// ── Aggregate readiness / faults ──────────────────────────────────────────────
allReady :=
    upperMasterReady AND upperSlave1VfdReady AND upperSlave2VfdReady AND
    lowerMasterReady AND lowerSlave1VfdReady AND lowerSlave2VfdReady;

anyFault :=
    groupFault OR
    upperMasterVfdFaultFeedback OR upperSlave1VfdFaultFeedback OR upperSlave2VfdFaultFeedback OR
    lowerMasterVfdFaultFeedback OR lowerSlave1VfdFaultFeedback OR lowerSlave2VfdFaultFeedback;

// ── Near-zero checks (unit must match your speed signals) ─────────────────────
speedsNearZero :=
    (ABS(upperMasterSpeedFeedback) <= speedZeroThresholdPct) AND
    (ABS(upperSlave1SpeedFeedback) <= speedZeroThresholdPct) AND
    (ABS(upperSlave2SpeedFeedback) <= speedZeroThresholdPct) AND
    (ABS(lowerMasterSpeedFeedback) <= speedZeroThresholdPct) AND
    (ABS(lowerSlave1SpeedFeedback) <= speedZeroThresholdPct) AND
    (ABS(lowerSlave2SpeedFeedback) <= speedZeroThresholdPct);

// Masters’ references near zero (backup condition)
refsNearZero :=
    (ABS(upperMasterDriveSpeedRefRPM) <= epsRefPct) AND
    (ABS(lowerMasterDriveSpeedRefRPM) <= epsRefPct);

// ── State machine ─────────────────────────────────────────────────────────────
CASE state OF
    0: // IDLE
        deviceState := 'IDLE';
        rampReset   := TRUE;

        // Ensure outputs are safe
        upperMasterDriveEnable := FALSE;
        upperSlave1DriveEnable := FALSE;
        upperSlave2DriveEnable := FALSE;
        lowerMasterDriveEnable := FALSE;
        lowerSlave1DriveEnable := FALSE;
        lowerSlave2DriveEnable := FALSE;

        IF rStart AND NOT anyFault THEN
            state := 1;
        END_IF

    1: // ENABLE_DRIVES
        deviceState := 'ENABLE_DRIVES';
        rampReset   := TRUE;

        // Enable all six drives
        upperMasterDriveEnable := TRUE;
        upperSlave1DriveEnable := TRUE;
        upperSlave2DriveEnable := TRUE;
        lowerMasterDriveEnable := TRUE;
        lowerSlave1DriveEnable := TRUE;
        lowerSlave2DriveEnable := TRUE;

        // Start enable wait timer
        instTONEnableWait(IN := TRUE, PT := enableTimeout);

        IF rStop OR stopGroup THEN
            instTONEnableWait(IN := FALSE);
            state := 5; // go to stopping
        ELSE
            state := 2; // proceed to wait feedback
        END_IF

    2: // WAIT_ENABLE_FEEDBACK
        deviceState := 'WAIT_ENABLE_FEEDBACK';
        rampReset   := TRUE;

        // Keep enables on while waiting
        upperMasterDriveEnable := TRUE;
        upperSlave1DriveEnable := TRUE;
        upperSlave2DriveEnable := TRUE;
        lowerMasterDriveEnable := TRUE;
        lowerSlave1DriveEnable := TRUE;
        lowerSlave2DriveEnable := TRUE;

        instTONEnableWait(IN := TRUE, PT := enableTimeout);

        IF anyFault THEN
            instTONEnableWait(IN := FALSE);
            state := 10; // FAULT
        ELSIF rStop OR stopGroup THEN
            instTONEnableWait(IN := FALSE);
            state := 5; // STOPPING
        ELSIF allReady THEN
            instTONEnableWait(IN := FALSE);
            state := 3; // RAMP_ENABLE
        ELSIF instTONEnableWait.Q THEN
            instTONEnableWait(IN := FALSE);
            state := 10; // fault: no enable feedback in time
        END_IF

    3: // RAMP_ENABLE (single-cycle gate to release ramp)
        deviceState := 'RAMP_ENABLE';
        rampReset   := FALSE; // release ramp now

        // Keep enables on
        upperMasterDriveEnable := TRUE;
        upperSlave1DriveEnable := TRUE;
        upperSlave2DriveEnable := TRUE;
        lowerMasterDriveEnable := TRUE;
        lowerSlave1DriveEnable := TRUE;
        lowerSlave2DriveEnable := TRUE;

        IF rStop OR stopGroup THEN
            state := 5;
        ELSE	
		
            state := 4; // RUN
					
        END_IF

    4: // RUN
        deviceState := SEL(groupSpeedAutoMan, 'RUN (Manual)', 'RUN (Auto)');
        rampReset   := FALSE;

        // Keep enables on during run
        upperMasterDriveEnable := TRUE;
        upperSlave1DriveEnable := TRUE;
        upperSlave2DriveEnable := TRUE;
        lowerMasterDriveEnable := TRUE;
        lowerSlave1DriveEnable := TRUE;
        lowerSlave2DriveEnable := TRUE;

        IF anyFault THEN
            state := 10; // FAULT
        ELSIF rStop OR stopGroup THEN
            state := 5;  // STOPPING
        END_IF

    5: // STOPPING (controlled decel)
        deviceState := 'STOPPING';
        rampReset   := FALSE; // allow ramp to drive refs down

        // Keep enables TRUE for controlled decel
        upperMasterDriveEnable := TRUE;
        upperSlave1DriveEnable := TRUE;
        upperSlave2DriveEnable := TRUE;
        lowerMasterDriveEnable := TRUE;
        lowerSlave1DriveEnable := TRUE;
        lowerSlave2DriveEnable := TRUE;

        // Optional: stop timeout (enable if you want a hard cutoff)
        // instTONStopWait(IN := TRUE, PT := stopTimeout);

        // Exit when speeds≈0 and refs≈0
        IF anyFault THEN
            // instTONStopWait(IN := FALSE);
            state := 10;

        ELSIF speedsNearZero AND refsNearZero THEN
            // Disable all drives
            upperMasterDriveEnable := FALSE;
            upperSlave1DriveEnable := FALSE;
            upperSlave2DriveEnable := FALSE;
            lowerMasterDriveEnable := FALSE;
            lowerSlave1DriveEnable := FALSE;
            lowerSlave2DriveEnable := FALSE;

            // instTONStopWait(IN := FALSE);
            state := 0; // IDLE

        ELSIF instTONStopWait.Q THEN
            // Timeout path → force disable then fault
            upperMasterDriveEnable := FALSE;
            upperSlave1DriveEnable := FALSE;
            upperSlave2DriveEnable := FALSE;
            lowerMasterDriveEnable := FALSE;
            lowerSlave1DriveEnable := FALSE;
            lowerSlave2DriveEnable := FALSE;

            instTONStopWait(IN := FALSE);
            state := 10;
        END_IF

    10: // FAULT
        deviceState := 'FAULT';
        rampReset   := TRUE; // force ramp outputs to zero

        // Disable all drives
        upperMasterDriveEnable := FALSE;
        upperSlave1DriveEnable := FALSE;
        upperSlave2DriveEnable := FALSE;
        lowerMasterDriveEnable := FALSE;
        lowerSlave1DriveEnable := FALSE;
        lowerSlave2DriveEnable := FALSE;

        // Return to IDLE when faults clear and start released
        IF (NOT anyFault) AND (NOT startGroup) THEN
            state := 0;
        END_IF
END_CASE
END_METHOD

// 2) REFERENCE GENERATOR
// Applies:
//   - groupSpeedOffset: added to ALL motors in this drying section (via ratio)
//   - uperAndLowerSpeedOffset: additional bias between UPPER and LOWER groups only
METHOD _ReferenceGenerator
VAR
    // ---------- Limits & helpers ----------
    headroomEpsPct      : REAL := 0.20;     // anti-chatter near saturation (100%)
    offsetPct           : REAL;             // slave speed offset as ratio (e.g., 10% -> 0.10)
    denom               : REAL;             // gear + offset denominator guard
    maxMasterBySlave    : REAL;             // master % at which a slave would hit 100%
    allowedCapPct       : REAL;             // master upward cap (prevents slave > 100%)
    cmdSpeedMPM         : REAL;             // selected command speed (m/min)
    targetRPM           : REAL;             // 0..100 scaled line reference before ramp

    // ---------- Freeze upward overrun ----------
    currMasterPct       : REAL;             // current ramp output for master (%)
    currSlavePct        : REAL;             // current synthetic slave (%), for freeze check

    // ---------- Group offsets ----------
    groupDeltaRatioAll  : REAL;             // = 1 + (groupSpeedOffset / 100) → applies to ALL motors
    upperLowerBiasRatio : REAL;             // = 1 + (uperAndLowerSpeedOffset / 100) → LOWER only

    // ---------- Convenience ----------
    baseMasterRefRPM    : REAL;             // common master reference after ramp/cap (pre-offsets)
    baseCmdSpeedMPM     : REAL;             // base command (auto/manual, pre-recover)

//	masterMaxSpeedMPM : REAL;

	PI : REAL := 3.14159265359;
	
	k_pi_per_1000 : REAL := 0.00314159265358979323846264338328;
	
END_VAR
//==============================================================
// Calculate max output speed in MPM
//==============================================================
masterMaxSpeedMPM := groupMasterMaxSpeedRPM * (PI * upperMasterDiameter) / 1000.0;


//==============================================================
// 1) Determine base speed source (auto or manual)
//==============================================================
IF groupSpeedAutoMan THEN
    baseCmdSpeedMPM := groupAutoSpeedMPM * interGroupGearRatio; // Auto reference (calibrated)
ELSE
    baseCmdSpeedMPM := groupManualSpeedMPM;                      // Manual reference (raw)
END_IF;


//==============================================================
// 2) Apply "Recover" temporary speed bump
//==============================================================
IF groupRecoverSpeedCmd THEN
    cmdSpeedMPM := baseCmdSpeedMPM + groupRecoverIncrement;     // Apply recover bump
ELSE
    cmdSpeedMPM := baseCmdSpeedMPM;                             // Normal operation
END_IF;


//==============================================================
// 3) Scale to target RPM for the drives 
//==============================================================
targetRPM := _Scale(
    X    := cmdSpeedMPM,
    I_LO := 0.0,          I_HI := masterMaxSpeedMPM,
    O_LO := 0.0,          O_HI := groupMasterMaxSpeedRPM);
	

//==============================================================
// 4) During STOPPING set target to 0 (still ramp down); otherwise track target
//==============================================================
IF state = 5 THEN
    rampTargetRPM := 0.0;
ELSE
    rampTargetRPM := targetRPM;
END_IF;


//==============================================================
// 5) Ramp (common line reference for this drying section)
//==============================================================
useRamp := (ABS(rampTargetRPM - instFB_Gen_SRamp.Y) >= 2.0);

instFB_Gen_SRamp(
    X          := rampTargetRPM,
    A_UP       := MAX(0.0, rampRate),
    A_DN       := -MAX(0.0, rampRate),
    VU_MAX     := 1000.0,
    VD_MAX     := -1000.0,
    LIMIT_HIGH := groupMasterMaxSpeedRPM,
    RST        := rampReset);

IF useRamp THEN
    baseMasterRefRPM := instFB_Gen_SRamp.Y;
ELSE
    baseMasterRefRPM := rampTargetRPM;
END_IF;


//==============================================================
// 6) Operator-adjustable groupSpeedOffset using TUNE2
//==============================================================
instTUNE2_GroupSpeedDiference(
    SET     := FALSE,
    SU      := groupSpeedDifInc,
    SD      := groupSpeedDifDec,
    RST     := FALSE,
    SS      := 0.1,
    FS      := 0.0,
    LIMIT_L := groupSpeedDifLimLow,
    LIMIT_H := groupSpeedDifLimHigh,
    Y       => groupSpeedOffset);

groupDeltaRatioAll  := 1.0 + (groupSpeedOffset * 0.01);
upperLowerBiasRatio := 1.0 + (upperAndLowerSpeedOffset * 0.01);


//==============================================================
// 7) MASTER references and slave ratios
//==============================================================
upperMasterDriveSpeedRefRPM := baseMasterRefRPM * groupDeltaRatioAll;

upperSlave1DriveSpeedRefRPM := upperMasterDriveSpeedRefRPM * upperToUpperSlave1Ratio;
upperSlave2DriveSpeedRefRPM := upperMasterDriveSpeedRefRPM * upperToUpperSlave2Ratio;

lowerMasterDriveSpeedRefRPM := upperMasterDriveSpeedRefRPM * upperToLowerMasterRatio;
lowerSlave1DriveSpeedRefRPM := lowerMasterDriveSpeedRefRPM * lowerToLowerSlave1Ratio;
lowerSlave2DriveSpeedRefRPM := lowerMasterDriveSpeedRefRPM * lowerToLowerSlave2Ratio;


//==============================================================
// 8) Convert drive RPM references to surface speeds in MPM
//==============================================================
upperMasterSpeedSetpointMPM := upperMasterDriveSpeedRefRPM * upperMasterDiameter * PI / 1000.0;
upperSlave1SpeedSetpointMPM := upperSlave1DriveSpeedRefRPM * upperSlave1Diameter * PI / 1000.0;
upperSlave2SpeedSetpointMPM := upperSlave2DriveSpeedRefRPM * upperSlave2Diameter * PI / 1000.0;

lowerMasterSpeedSetpointMPM := lowerMasterDriveSpeedRefRPM * lowerMasterDiameter * PI / 1000.0;
lowerSlave1SpeedSetpointMPM := lowerSlave1DriveSpeedRefRPM * lowerSlave1Diameter * PI / 1000.0;
lowerSlave2SpeedSetpointMPM := lowerSlave2DriveSpeedRefRPM * lowerSlave2Diameter * PI / 1000.0;
END_METHOD

METHOD PRIVATE _Scale : REAL
VAR_INPUT
    X    : REAL;
    I_LO : REAL;
    I_HI : REAL;
    O_LO : REAL;
    O_HI : REAL;
END_VAR
IF I_LO = I_HI THEN
	_Scale := O_LO;
ELSE
	_Scale := (O_HI - O_LO) / (I_HI - I_LO) * (LIMIT(I_LO, X, I_HI) - I_LO) + O_LO;
END_IF;
END_METHOD

METHOD PRIVATE _SpeedDifferenceCheck
VAR
    diffUpper : REAL; // max |Master - Slave| in UPPER group
    diffLower : REAL; // max |Master - Slave| in LOWER group
    diffMax   : REAL; // worst-case across both groups
END_VAR

(*
// ── Compare only within each group: Master ↔ Slaves (ignore cross-group) ──────
// UPPER group (Master vs Slave1, Master vs Slave2)
diffUpper :=
    MAX(
        ABS(upperMasterSpeedMPMFilteredDisplay - upperSlave1SpeedMPMFilteredDisplay),
        ABS(upperMasterSpeedMPMFilteredDisplay - upperSlave2SpeedMPMFilteredDisplay)
    );

// LOWER group (Master vs Slave1, Master vs Slave2)
diffLower :=
    MAX(
        ABS(lowerMasterSpeedMPMFilteredDisplay - lowerSlave1SpeedMPMFilteredDisplay),
        ABS(lowerMasterSpeedMPMFilteredDisplay - lowerSlave2SpeedMPMFilteredDisplay)
    );

// Pick worst intra-group deviation and expose for diagnostics/HMI
diffMax := MAX(diffUpper, diffLower);
currentSpeedDifence := diffMax;

// ── Trip logic with delay (debounce) ───────────────────────────────────────────
instTONSpeedDifDelay(
    IN := (diffMax > speedDiferenceLimit),
    PT := T#2s
);

IF instTONSpeedDifDelay.Q THEN
    state := 10; // FAULT
    deviceState := 'FAULT: Intra-group speed difference exceeded';
END_IF
*)
END_METHOD

METHOD _StateDisplay
VAR_INPUT
END_VAR

// ──────────────────────────────────────────────────────────────────────────────
// _StateDisplay
// Maps the internal machine "state" to a compact HMI status code and derives
// per-drive motor status codes from VFD signals.
//
// statusCode / masterStatusCode / slaveStatusCode legend:
//   0 = Idle, 1 = Starting, 2 = Running, 3 = Fault
//
// Machine "state" groups:
//   0 = IDLE, 1 = ENABLE, 2 = WAIT_EN, 3 = RAMP_EN, 4 = RUN, 5 = STOPPING, 10 = FAULT
// Priority rule (for motors): Fault > Running > Starting > Idle
// ──────────────────────────────────────────────────────────────────────────────
VAR CONSTANT
    STATUS_IDLE     : INT := 0;
    STATUS_STARTING : INT := 1;
    STATUS_RUNNING  : INT := 1;
    STATUS_FAULT    : INT := 2;
END_VAR
// ─────────────── Group machine states into a single HMI statusCode ───────────
CASE state OF
    10: // FAULT
        statusCode := STATUS_FAULT;
    4:  // RUN
        statusCode := STATUS_RUNNING;
    1, 2, 3: // ENABLE / WAIT_EN / RAMP_EN
        statusCode := STATUS_STARTING;
ELSE // IDLE, STOPPING, or any other
        statusCode := STATUS_IDLE;
END_CASE;


// ─────────────── Per-drive status (priority: Fault > Running > Starting > Idle) ───────────────
// UPPER — MASTER
IF upperMasterVfdFaultFeedback THEN
    upperMasterStatusCode := STATUS_FAULT;
ELSIF upperMasterVfdRunFeedback THEN
    upperMasterStatusCode := STATUS_RUNNING;
ELSIF upperMasterDriveEnable THEN
    upperMasterStatusCode := STATUS_STARTING;
ELSE
    upperMasterStatusCode := STATUS_IDLE;
END_IF;

// UPPER — SLAVE 1
IF upperSlave1VfdFaultFeedback THEN
    upperSlave1StatusCode := STATUS_FAULT;
ELSIF upperSlave1VfdRunFeedback THEN
    upperSlave1StatusCode := STATUS_RUNNING;
ELSIF upperSlave1DriveEnable THEN
    upperSlave1StatusCode := STATUS_STARTING;
ELSE
    upperSlave1StatusCode := STATUS_IDLE;
END_IF;

// UPPER — SLAVE 2
IF upperSlave2VfdFaultFeedback THEN
    upperSlave2StatusCode := STATUS_FAULT;
ELSIF upperSlave2VfdRunFeedback THEN
    upperSlave2StatusCode := STATUS_RUNNING;
ELSIF upperSlave2DriveEnable THEN
    upperSlave2StatusCode := STATUS_STARTING;
ELSE
    upperSlave2StatusCode := STATUS_IDLE;
END_IF;

// LOWER — MASTER
IF lowerMasterVfdFaultFeedback THEN
    lowerMasterStatusCode := STATUS_FAULT;
ELSIF lowerMasterVfdRunFeedback THEN
    lowerMasterStatusCode := STATUS_RUNNING;
ELSIF lowerMasterDriveEnable THEN
    lowerMasterStatusCode := STATUS_STARTING;
ELSE
    lowerMasterStatusCode := STATUS_IDLE;
END_IF;

// LOWER — SLAVE 1
IF lowerSlave1VfdFaultFeedback THEN
    lowerSlave1StatusCode := STATUS_FAULT;
ELSIF lowerSlave1VfdRunFeedback THEN
    lowerSlave1StatusCode := STATUS_RUNNING;
ELSIF lowerSlave1DriveEnable THEN
    lowerSlave1StatusCode := STATUS_STARTING;
ELSE
    lowerSlave1StatusCode := STATUS_IDLE;
END_IF;

// LOWER — SLAVE 2
IF lowerSlave2VfdFaultFeedback THEN
    lowerSlave2StatusCode := STATUS_FAULT;
ELSIF lowerSlave2VfdRunFeedback THEN
    lowerSlave2StatusCode := STATUS_RUNNING;
ELSIF lowerSlave2DriveEnable THEN
    lowerSlave2StatusCode := STATUS_STARTING;
ELSE
    lowerSlave2StatusCode := STATUS_IDLE;
END_IF;
END_METHOD

METHOD _SteamPressureControl
VAR_INPUT
END_VAR

//────────────────────────────────────────────────────────────
// PID — Steam Pressure Control
//────────────────────────────────────────────────────────────
instCTRL_PID_TemperatureController(
    ACT := steamPressureFeedback,                          // Real-time feedback (PV)
    SET := SEL(steamPressureAutoMan,                       // Setpoint selection
               steamPressureManualSetpoint,                // Manual setpoint
               steamPressureAutoSetpoint),                 // Auto setpoint
    MAN := steamPressureAutoMan = FALSE,                   // Manual mode when AutoMan is FALSE
    M_I := steamPressureManualSetpoint,                    // Tracks manual setpoint
    RST := FALSE,                                          // No reset
    KP  := steamPressureKp,                               
    TN  := steamPressureTn,                               
    TV  := steamPressureTv,                               
    LL  := 0.0,                                            // Output lower limit
    LH  := 100.0,                                          // Output upper limit [%]
    Y   => steamPressureControllerOutput                   // PID output
);
END_METHOD

METHOD PRIVATE _TorqueReference
VAR
    // UPPER
    rawTorqueUpper      : REAL;
    filteredTorqueUpper : REAL;
    capMasterUpper      : REAL; // ≤ master, ≤ global max
    baseLimitUpper      : REAL; // (master + offset) capped by master
    directTorqueUpper   : REAL; // direct write portion
    avgTorqueUpper      : REAL;
    trimUp              : REAL; // PID top-up (≥0)

    // LOWER
    rawTorqueLower      : REAL;
    filteredTorqueLower : REAL;
    capMasterLower      : REAL;
    baseLimitLower      : REAL;
    directTorqueLower   : REAL;
    avgTorqueLower      : REAL;
    trimLo              : REAL;
END_VAR


// ── UPPER ─────────────────────────────────────────────────────────────────────
rawTorqueUpper := upperMasterTorqueFeedback;
instsFT_PT1UpperTorqueFilter( in := rawTorqueUpper, 
							   T := torqueFilterTime, 
							   K := 1.0, 
							   out => filteredTorqueUpper );
							   

// Master cap and base limit (never exceed master)
capMasterUpper := LIMIT(torqueLimitMinPct, filteredTorqueUpper, torqueLimitMaxPct);
baseLimitUpper := MIN(
    capMasterUpper,
    LIMIT(torqueLimitMinPct, filteredTorqueUpper + slaveTorqueOfsset, torqueLimitMaxPct)
);

IF NOT enableTorquePid THEN
    upperSlave1DriveTorqueRefPct := capMasterUpper;
    upperSlave2DriveTorqueRefPct := capMasterUpper;
ELSE
    directTorqueUpper := LIMIT(torqueLimitMinPct, baseLimitUpper - torqueTrimLimit, capMasterUpper);
    avgTorqueUpper    := 0.5 * (upperSlave1TorqueFeedback + upperSlave2TorqueFeedback);

    instCTRL_PID_UpperTorqueTrim(
        ACT := avgTorqueUpper,
        SET := baseLimitUpper,
        MAN := NOT enableTorquePid,   // manual when disabled (tracks 0)
        M_I := 0.0,
        RST := FALSE,
        KP  := torqueCtrlKp,
        TN  := torqueCtrlTn,
        TV  := torqueCtrlTv,
        LL  := 0.0,                   // unipolar: only add
        LH  := torqueTrimLimit,
        Y   => trimUp
    );

    upperSlave1DriveTorqueRefPct := LIMIT(torqueLimitMinPct, directTorqueUpper + trimUp, capMasterUpper);
    upperSlave2DriveTorqueRefPct := LIMIT(torqueLimitMinPct, directTorqueUpper + trimUp, capMasterUpper);
END_IF;


// ── LOWER ─────────────────────────────────────────────────────────────────────
rawTorqueLower := lowerMasterTorqueFeedback;
instsFT_PT1LowerTorqueFilter( in := rawTorqueLower, T := torqueFilterTime, K := 1.0, out => filteredTorqueLower );

capMasterLower := LIMIT(torqueLimitMinPct, filteredTorqueLower, torqueLimitMaxPct);
baseLimitLower := MIN(
    capMasterLower,
    LIMIT(torqueLimitMinPct, filteredTorqueLower + slaveTorqueOfsset, torqueLimitMaxPct)
);

IF NOT enableTorquePid THEN
    lowerSlave1DriveTorqueRefPct := capMasterLower;
    lowerSlave2DriveTorqueRefPct := capMasterLower;
ELSE
    directTorqueLower := LIMIT(torqueLimitMinPct, baseLimitLower - torqueTrimLimit, capMasterLower);
    avgTorqueLower    := 0.5 * (lowerSlave1TorqueFeedback + lowerSlave2TorqueFeedback);

    instCTRL_PID_LowerTorqueTrim(
        ACT := avgTorqueLower,
        SET := baseLimitLower,
        MAN := NOT enableTorquePid,
        M_I := 0.0,
        RST := FALSE,
        KP  := torqueCtrlKp,
        TN  := torqueCtrlTn,
        TV  := torqueCtrlTv,
        LL  := 0.0,
        LH  := torqueTrimLimit,
        Y   => trimLo
    );

    lowerSlave1DriveTorqueRefPct := LIMIT(torqueLimitMinPct, directTorqueLower + trimLo, capMasterLower);
    lowerSlave2DriveTorqueRefPct := LIMIT(torqueLimitMinPct, directTorqueLower + trimLo, capMasterLower);
END_IF;


// ── Safety (optional) ─────────────────────────────────────────────────────────
IF (state < 3) OR (state = 5) OR (state = 10) THEN
    upperSlave1DriveTorqueRefPct := 0.0;
    upperSlave2DriveTorqueRefPct := 0.0;
    lowerSlave1DriveTorqueRefPct := 0.0;
    lowerSlave2DriveTorqueRefPct := 0.0;
END_IF
END_METHOD

END_FUNCTION_BLOCK

// ---- Function Blocks/Rewinder/FB_RewinderControl_V1.TcPOU
FUNCTION_BLOCK FB_RewinderControl_V1
VAR_INPUT

    //==============================================================
    // ─────────────── BASIC COMMANDS / MACHINE INTERFACE ───────────────
    //==============================================================
    startCmd                    : BOOL;  // EN: Start rewinder command / PT: Comando de partida do rebobinador
    stopCmd                     : BOOL;  // EN: Stop rewinder command / PT: Comando de parada do rebobinador
	
	jogCmd						: BOOL;
  
	rewinderAutoMan            : BOOL;  // EN: Auto/Manual selector (FALSE = Manual) / PT: Seletor Auto/Manual (FALSE = Manual)

	
	rollEjectorFwCmd			: BOOL;
	rollEjectorRevCmd			: BOOL;
	
	
	
    //==============================================================
    // ─────────────── SPEED MONITORING / LIMITS ───────────────
    //==============================================================
    speedFeedBackMPM           : REAL;  // EN: Actual machine speed [m/min] / PT: Velocidade atual da máquina [m/min]
    groupMaxSpeed              : REAL;  // EN: Max allowed speed [m/min] / PT: Velocidade máxima permitida [m/min]

    //==============================================================
    // ─────────────── PRESS ROLL / NIP CONTROL ───────────────
    //==============================================================
    pressRollAutoMan           : BOOL;  // EN: Press roll Auto/Manual selector (FALSE = Manual) / PT: Seletor Auto/Manual do rolo de pressão (FALSE = Manual)
  
    pressRollManualSetpoint    : REAL;  // EN: Manual press roll setpoint / PT: Setpoint manual de posição/pressão do rolo de pressão
    //==============================================================
    // ─────────────── PRESS ROLL / NIP OUTPUTS ───────────────
    //==============================================================

    pressRollCmdUp             : BOOL;  // EN: Output command to open press roll / PT: Comando de abertura do rolo de pressão
    pressRollCmdDown           : BOOL;  // EN: Output command to close press roll / PT: Comando de fechamento do rolo de pressão

    //==============================================================
    // ─────────────── DIAMETER INPUTS ───────────────
    //==============================================================
    rewinderRollDiameter       : REAL;  // EN: Rewinder roll (winding) diameter [mm] / PT: Diâmetro do rolo rebobinado [mm]
    unwinderRollDiameter       : REAL;  // EN: Unwinder roll (payoff) diameter [mm] / PT: Diâmetro do rolo desbobinado [mm]

    //==============================================================
    // ─────────────── TENSION CONTROL ───────────────
    //==============================================================
    tensionSetpointN           : REAL;  // EN: Web tension setpoint [N] / PT: Setpoint de tensão da folha [N]
    tensionFeedbackN           : REAL;  // EN: Web tension feedback from load cell [N] / PT: Leitura de tensão da célula de carga [N]
    tensionControlEnable       : BOOL;  // EN: Enable tension control / PT: Habilita controle de tensão

    //==============================================================
    // ─────────────── ROLL LIMITS ───────────────
    //==============================================================
    maxRewinderDiameter        : REAL;  // EN: Max rewinder roll diameter [mm] / PT: Diâmetro máximo do rebobinador [mm]

    //==============================================================
    // ─────────────── SAFETY / INTERLOCKS ───────────────
    //==============================================================
    safetyCircuitOK            : BOOL;  // EN: Safety circuit healthy / PT: Circuito de segurança OK
    webBreakSensor             : BOOL;  // EN: Web break sensor triggered / PT: Sensor de ruptura de folha

    //==============================================================
    // ─────────────── SPEED REFERENCE INPUTS ───────────────
    //==============================================================
    rewinderAutoSpeedRefMPM    : REAL;  // EN: Auto speed reference (external) [m/min] / PT: Referência automática de velocidade [m/min]
    rewinderManualSpeedRefMPM  : REAL;  // EN: Manual speed reference [m/min] / PT: Referência manual de velocidade [m/min]
    rampRate                   : REAL := 0.01;  // EN: Ramp acceleration rate [%/s] / PT: Taxa de aceleração da rampa [%/s]
	
	
    //==============================================================
    // ─────────────── WEB GUIDING / EDGE CONTROL ───────────────
    //==============================================================
    unwinderRollOperatorSideCmd   : BOOL;  // EN: Operator-side web guide control / PT: Controle de guia lado operador
    unwinderRollDriveSideCmd      : BOOL;  // EN: Drive-side web guide control / PT: Controle de guia lado acionamento
	unwinderRollOperatorSideLimitSensor   : BOOL;  // EN: Operator-side web guide control / PT: Controle de guia lado operador
    unwinderRollDriveSideLimitSensor      : BOOL;  // EN: Drive-side web guide control / PT: Controle de guia lado acionamento
    unwinderShaftLockedSensor      		: BOOL;  // EN: Drive-side web guide control / PT: Controle de guia lado acionamento
    unwinderRollBrakeCoupledSensor      : BOOL;  // EN: Drive-side web guide control / PT: Controle de guia lado acionamento
	
   rewinderCoreClampSolenoidCmd : BOOL;   // EN: Solenoid valve command to lock (clamp) the core of the rewinding roll / PT: Comando da válvula solenóide que trava o tubete (manga) do rolo em enrolamento

	// ─────────────── ROLL CHUTE / BIN INPUTS ───────────────
	rollBinAtLoadPositionSensor     : BOOL;   // EN: Sensor — bin/chute at load position / PT: Sensor — caçamba na posição de carga	
	rollBinAtUnloadPositionSensor   : BOOL;   // EN: Sensor — bin/chute at unload position / PT: Sensor — caçamba na posição de descarte
	rollBinRequestUnloadPosCmd      : BOOL;   // EN: Command to trigger bin unloading / PT: Comando para iniciar descarregamento da caçamba	
	rollBinRequestLoadPosCmd      : BOOL;   // EN: Command to trigger bin unloading / PT: Comando para iniciar descarregamento da caçamba	
	rollBinSafetySensor     : BOOL;   // EN: Command to trigger bin unloading / PT: Comando para iniciar descarregamento da caçamba	
   
   machineConfig				: RewinderConfig_TypeStruct;
   

END_VAR

VAR_OUTPUT

	deviceState				: STRING;

    rewinderRollDiameterFiltered       : REAL;  // EN: Rewinder roll (winding) diameter [mm] / PT: Diâmetro do rolo rebobinado [mm]
    unwinderRollDiameterFiltered       : REAL;  // EN: Unwinder roll (payoff) diameter [mm] / PT: Diâmetro do rolo desbobinado [mm]

    //==============================================================
    // ─────────────── REWINDER DRIVE OUTPUTS ───────────────
    //==============================================================
    rewinderMotorStart         : BOOL;  // EN: Start/enable command for rewinder drive / PT: Comando de habilitação do motor rebobinador
    rewinderMotorSpeedRefMPM   : REAL;  // EN: Speed reference [m/min] / PT: Referência de velocidade [m/min]
    rewinderMotorSpeedRefPct   : REAL;  // EN: Speed/torque reference [%] / PT: Referência de velocidade/torque [%]


    //==============================================================
    // ─────────────── UNWINDER BRAKE OUTPUT ───────────────
    //==============================================================
    brakeSetpointPct           : REAL;  // EN: Unwinder brake setpoint [%] / PT: Setpoint do freio do desbobinador [%]

    //==============================================================
    // ─────────────── WEB GUIDING / EDGE CONTROL ───────────────
    //==============================================================
    unwinderRollOperatorSide   : BOOL;  // EN: Operator-side web guide control / PT: Controle de guia lado operador
    unwinderRollDriveSide      : BOOL;  // EN: Drive-side web guide control / PT: Controle de guia lado acionamento
	
	ressRollUP                : BOOL;  // EN: Command to lift/open press roll / PT: Comando para levantar/abrir o rolo de pressão
    pressRollDown              : BOOL;  // EN: Command to lower/close press roll / PT: Comando para descer/fechar o rolo de pressão  
	pressRollSetpoint          : REAL;  // EN: Final press roll setpoint / PT: Setpoint final do rolo de pressão
	rewinderCoreClampSolenoid : BOOL;   // EN: Solenoid valve command to lock (clamp) the core of the rewinding roll / PT: Comando da válvula solenóide que trava o tubete (manga) do rolo em enrolamento

	
	rollEjectorFw			: BOOL;
	rollEjectorRev			: BOOL;
	
	rollBinRequestUnloadPos      : BOOL;   // EN: Command to trigger bin unloading / PT: Comando para iniciar descarregamento da caçamba	
	rollBinRequestLoadPos      : BOOL;   // EN: Command to trigger bin unloading / PT: Comando para iniciar descarregamento da caçamba	
			
	
END_VAR

VAR

    i                      : INT;
    x0, x1, y0, y1         : REAL;
    interpOutput           : REAL;

	firstCycle		: BOOL := TRUE;
    //==============================================================
    // ─────────────── RAMP BLOCK / REFERENCES ───────────────
    //==============================================================
    instFB_Gen_SRamp           : FB_Gen_SRamp; // EN: S-curve ramp function block / PT: Bloco de rampa S
	
    instFB_Gen_SRampPressRoll           : FB_Gen_SRamp; // EN: S-curve ramp function block / PT: Bloco de rampa S
    instFB_Gen_SRampBrake           	: FB_Gen_SRamp; // EN: S-curve ramp function block / PT: Bloco de rampa S
	
	
    rampTargetPct              : REAL;         // EN: Target % reference for ramp / PT: Referência alvo [%] para a rampa
    rampReset                  : BOOL;         // EN: Ramp reset command / PT: Comando de reset da rampa

    //==============================================================
    // ─────────────── INTERNAL STATE / EDGE DETECT ───────────────
    //==============================================================
    rewinderState              : INT;          // EN: Main state (0=IDLE .. 5=STOPPING .. 10=FAULT) / PT: Estado principal (0=IDLE .. 5=PARANDO .. 10=FALHA)
    startCmdOld                : BOOL;
    stopCmdOld                 : BOOL;
    rStart                     : BOOL;         // EN: Rising edge detector for start / PT: Borda de subida para partida
    rStop                      : BOOL;         // EN: Rising edge detector for stop / PT: Borda de subida para parada
//    state                      : INT;

    //==============================================================
    // ─────────────── TIMERS ───────────────
    //==============================================================
    tonEnableWait              : TON;          // EN: Delay after enable / PT: Retardo após habilitação
    tonStopWait                : TON;          // EN: Delay after stop / PT: Retardo após parada
    enableTimeout              : TIME := T#5S;
    stopTimeout                : TIME := T#8S;

    //==============================================================
    // ─────────────── LOGIC CONDITIONS ───────────────
    //==============================================================
    anyFault                   : BOOL;         // EN: Any fault detected / PT: Alguma falha presente
    speedsNearZero             : BOOL;         // EN: TRUE if speed below threshold / PT: Verdadeiro se velocidade for baixa
    refsNearZero               : BOOL;         // EN: TRUE if reference near zero / PT: Verdadeiro se referência for próxima de zero
    speedZeroThresholdMPM      : REAL := 3.0;  // EN: Below this = zero speed / PT: Abaixo disso considera parado
    epsRefMPM                  : REAL := 0.5;  // EN: Small epsilon for speed reference / PT: Margem mínima para referência de velocidade

    //==============================================================
    // ─────────────── FEEDBACKS ───────────────
    //==============================================================
    rewinderReadyFeedback      : BOOL;         // EN: Ready signal from drive / PT: Sinal de pronto do inversor

	rollEjectorFwCmdOld			: BOOL;
	
	  rRollEjectorFwCmd : BOOL; // Rising edge for forward
	  
	  
    // ---------- Limits & helpers ----------
    headroomEpsPct      : REAL := 0.20;     // anti-chatter near saturation (100%)
    allowedCapPct       : REAL;             // master upward cap (prevents >100%)
    cmdSpeedMPM         : REAL;             // selected command speed (m/min)
    targetPct           : REAL;             // 0..100 scaled reference before ramp
    currMasterPct       : REAL;             // current ramp output (%)
    baseCmdSpeedMPM     : REAL;             // base command (auto/manual)
	
//    speedsNearZero  : BOOL;  // EN: Speed near zero / PT: Velocidade próxima de zero
 //   refsNearZero    : BOOL;  // EN: Reference near zero / PT: Referência próxima de zero
//    anyFault        : BOOL;  // EN: Fault condition / PT: Condição de falha
    allReady        : BOOL;  // EN: Ready feedback OK / PT: Drive pronto		  
	  
END_VAR


_GroupControl();
_PressRollControl();
_ReferenceGenerator();
_rollBinControl();
_RollEjectorControl();


firstCycle		 := FALSE;

// ============================== Methods ==============================
// 1) GROUP CONTROL
METHOD _GroupControl
VAR_INPUT
END_VAR
VAR

END_VAR
// ──────────────────────────── Edge Detection ─────────────────────────────
rStart := startCmd AND NOT startCmdOld; // Pulse edge
rStop  := stopCmd  AND NOT stopCmdOld;
startCmdOld := startCmd;
stopCmdOld  := stopCmd;

// ──────────────────────────── Conditions ─────────────────────────────
allReady   := rewinderReadyFeedback AND safetyCircuitOK AND NOT webBreakSensor;
anyFault   := NOT safetyCircuitOK OR webBreakSensor;
//speedsNearZero := (ABS(speedFeedBackMPM) <= speedZeroThresholdMPM);
speedsNearZero :=  (ABS(rewinderMotorSpeedRefMPM) <= epsRefMPM);

refsNearZero   := (ABS(rewinderMotorSpeedRefMPM) <= epsRefMPM);

// ──────────────────────────── State Machine ─────────────────────────────
CASE rewinderState OF

    0: // IDLE
        deviceState := 'IDLE';
        rampReset := TRUE;

        rewinderMotorStart := FALSE;

        IF jogCmd AND NOT anyFault THEN
            rewinderState := 100; // Go to JOG
        ELSIF rStart AND NOT anyFault THEN
            rewinderState := 1;
        END_IF

    1: // ENABLE
        deviceState := 'ENABLE';
        rampReset := TRUE;

        rewinderMotorStart := TRUE;
        tonEnableWait(IN := TRUE, PT := enableTimeout);

        IF rStop OR stopCmd THEN
            tonEnableWait(IN := FALSE);
            rewinderState := 5;
        ELSE
            rewinderState := 2;
        END_IF

    2: // WAIT_FEEDBACK
        deviceState := 'WAIT_FEEDBACK';
        rampReset := TRUE;

        rewinderMotorStart := TRUE;
        tonEnableWait(IN := TRUE, PT := enableTimeout);

        IF anyFault THEN
            tonEnableWait(IN := FALSE);
            rewinderState := 10;

        ELSIF rStop OR stopCmd THEN
            tonEnableWait(IN := FALSE);
            rewinderState := 5;

        ELSIF allReady THEN
            tonEnableWait(IN := FALSE);
            rewinderState := 3;

        ELSIF tonEnableWait.Q THEN
            tonEnableWait(IN := FALSE);
            rewinderState := 10; // Fault: no feedback
        END_IF

    3: // RAMP_RELEASE
        deviceState := 'RAMP_RELEASE';
        rampReset := FALSE; // Release ramp
        rewinderMotorStart := TRUE;

        rewinderState := 4;

    4: // RUN
        deviceState := SEL(rewinderAutoMan, 'RUN (Auto)', 'RUN (Manual)');
        rampReset := FALSE;
        rewinderMotorStart := TRUE;

        IF anyFault THEN
            rewinderState := 10;
        ELSIF rStop OR stopCmd THEN
            rewinderState := 5;
        END_IF

    5: // STOPPING
        deviceState := 'STOPPING';
        rampReset := FALSE;
        rewinderMotorStart := TRUE;

        IF anyFault THEN
            rewinderState := 10;
        ELSIF speedsNearZero AND refsNearZero THEN
            rewinderMotorStart := FALSE;
            rewinderState := 0;
        ELSIF tonStopWait.Q THEN
            rewinderMotorStart := FALSE;
            tonStopWait(IN := FALSE);
            rewinderState := 10;
        END_IF

    10: // FAULT
        deviceState := 'FAULT';
        rampReset := TRUE;
        rewinderMotorStart := FALSE;

        IF (NOT anyFault) AND (NOT startCmd) THEN
            rewinderState := 0;
        END_IF

    100: // JOG MODE (Immediate Start)
        deviceState := 'JOG';
        rampReset := TRUE;
        rewinderMotorStart := TRUE;

        IF NOT jogCmd OR anyFault THEN
            rewinderMotorStart := FALSE;
            rewinderState := 0; // Back to IDLE when released or fault
        END_IF
END_CASE
END_METHOD

METHOD _PressRollControl
VAR

END_VAR

// Seleciona a referência base
IF pressRollAutoMan THEN
    // ─────── MODO AUTOMÁTICO ───────
    rewinderRollDiameterFiltered := rewinderRollDiameter;

    // Busca o intervalo para interpolação linear
    FOR i := 0 TO 18 DO
        IF rewinderRollDiameterFiltered >= machineConfig.arrPressRollParameters[i].rollDiameter AND
           rewinderRollDiameterFiltered <= machineConfig.arrPressRollParameters[i+1].rollDiameter THEN

            x0 := machineConfig.arrPressRollParameters[i].rollDiameter;
            y0 := machineConfig.arrPressRollParameters[i].pressureSetpoint;
            x1 := machineConfig.arrPressRollParameters[i+1].rollDiameter;
            y1 := machineConfig.arrPressRollParameters[i+1].pressureSetpoint;

            // Interpolação linear
            IF x1 <> x0 THEN
                interpOutput := y0 + (rewinderRollDiameterFiltered - x0) * (y1 - y0) / (x1 - x0);
            ELSE
                interpOutput := y0; // fallback (evita divisão por zero)
            END_IF;

            EXIT; // intervalo encontrado
        END_IF
    END_FOR
ELSE
    // ─────── MODO MANUAL ───────
    interpOutput := pressRollManualSetpoint;
END_IF

// ─────── Aplica rampa para suavizar o valor final ───────
instFB_Gen_SRampPressRoll(
    X := interpOutput,
    A_UP := 5.0,     // aceleração [unit/s] — pode ajustar
    A_DN := -5.0,    // desaceleração [unit/s]
    VU_MAX := 1000.0,
    VD_MAX := -1000.0,
    LIMIT_HIGH := 100.0,
    LIMIT_LOW := 0.0,
    RST := FALSE
);

// ─────── Seta a saída final ───────
pressRollSetpoint := instFB_Gen_SRampPressRoll.Y;
END_METHOD

//==============================================================
// REWINDER — SIMPLE SPEED REFERENCE GENERATOR
// EN: Generates the speed reference (% and m/min) for the rewinder motor
// PT: Gera a referência de velocidade (% e m/min) para o motor do rebobinador
//==============================================================
METHOD _ReferenceGenerator
VAR

END_VAR
//==============================================================
// 1) Determine base speed source (auto or manual)
//==============================================================
IF rewinderAutoMan THEN
    baseCmdSpeedMPM := rewinderManualSpeedRefMPM;   // Auto mode — follow main line
ELSE
    baseCmdSpeedMPM := rewinderAutoSpeedRefMPM;     // Manual mode — use local reference
END_IF;

//==============================================================
// 2) Apply stop condition and bin constraint
//==============================================================
IF rewinderState = 5 THEN
    cmdSpeedMPM := 0.0;
ELSIF rewinderState = 100 THEN
    // JOG MODE — direct jog reference
    cmdSpeedMPM := machineConfig.rewinderJogSpeedRefMPM;
ELSE
    // Normal operation — but limit to jog speed if bin not in load position
    cmdSpeedMPM := baseCmdSpeedMPM;

    IF NOT rollBinAtLoadPositionSensor THEN
        cmdSpeedMPM := MIN(cmdSpeedMPM, machineConfig.rewinderJogSpeedRefMPM);
    END_IF;
END_IF;

//==============================================================
// 3) Scale command speed to percentage (0–100%)
//==============================================================
targetPct := _Scale(
    X    := cmdSpeedMPM,
    I_LO := 0.0,
    I_HI := groupMaxSpeed,
    O_LO := 0.0,
    O_HI := 100.0);

//==============================================================
// 4) Limit and ramp
//==============================================================
allowedCapPct := 100.0;
rampTargetPct := LIMIT(0.0, MIN(targetPct, allowedCapPct), 100.0);

// Anti-chatter: freeze ramp up if near saturation
currMasterPct := instFB_Gen_SRamp.Y;
IF currMasterPct >= 100.0 - headroomEpsPct THEN
    rampTargetPct := MIN(rampTargetPct, currMasterPct);
END_IF;

//==============================================================
// 5) Ramp the command (smooth accel/decel)
//==============================================================
instFB_Gen_SRamp(
    X          := rampTargetPct,
    A_UP       := MAX(0.0, rampRate),
    A_DN       := -MAX(0.0, rampRate),
    VU_MAX     := 1000.0,
    VD_MAX     := -1000.0,
    LIMIT_HIGH := 100.0,
    RST        := rampReset);

IF rewinderState = 5 THEN
    instFB_Gen_SRamp.LIMIT_LOW := 0.0;
ELSE
    instFB_Gen_SRamp.LIMIT_LOW := 3.5;
END_IF;

//==============================================================
// 6) Final References
//==============================================================
IF rewinderState = 100 THEN // JOG
    rewinderMotorSpeedRefMPM := machineConfig.rewinderJogSpeedRefMPM;
    rewinderMotorSpeedRefPct := _Scale(
        X := machineConfig.rewinderJogSpeedRefMPM,
        I_LO := 0.0,
        I_HI := groupMaxSpeed,
        O_LO := 0.0,
        O_HI := 100.0);
ELSE
    // Normal ramped reference (possibly clamped by jog speed if bin not in place)
    rewinderMotorSpeedRefMPM := _Scale(
        X    := instFB_Gen_SRamp.Y,
        I_LO := 0.0,
        I_HI := 100.0,
        O_LO := 0.0,
        O_HI := groupMaxSpeed);
    rewinderMotorSpeedRefPct := instFB_Gen_SRamp.Y;
END_IF;
END_METHOD

METHOD _rollBinControl
VAR_INPUT
END_VAR
//==============================================================
// ROLL BIN CONTROL LOGIC
//==============================================================

// ──────────────────────────────
// SAFETY INTERLOCK — stop all movement
// ──────────────────────────────
IF rollBinSafetySensor OR firstCycle THEN
    rollBinRequestLoadPos := FALSE;
    rollBinRequestUnloadPos := FALSE;
ELSE
    // ──────────────────────────────
    // Move to LOAD position
    // ──────────────────────────────
    IF rollBinRequestLoadPosCmd THEN
        rollBinRequestLoadPos := TRUE;
	    rollBinRequestUnloadPos := FALSE;
	
    END_IF;

    // ──────────────────────────────
    // Move to UNLOAD position
    // ──────────────────────────────
    IF rollBinRequestUnloadPosCmd AND (rewinderState = 0) THEN
        rollBinRequestUnloadPos := TRUE;
	    rollBinRequestLoadPos := FALSE;
		
    END_IF;
END_IF;
END_METHOD

METHOD _RollEjectorControl
VAR_INPUT
END_VAR
//────────────────────────────────────────────────────────────
// Edge detection — borda de subida do comando de avanço
//────────────────────────────────────────────────────────────
rRollEjectorFwCmd := rollEjectorFwCmd AND NOT rollEjectorFwCmdOld;

//────────────────────────────────────────────────────────────
// Lógica de controle com intertravamentos
//────────────────────────────────────────────────────────────

// Condições para permitir avanço:
IF rRollEjectorFwCmd AND (rewinderState = 0) AND // Máquina parada (IDLE)
      rollBinAtLoadPositionSensor THEN
    // Prioridade para reversão
    rollEjectorFw := TRUE;
END_IF


IF rollEjectorRevCmd THEN
	
    rollEjectorFw := FALSE;

END_IF

rollEjectorFwCmdOld := rollEjectorFwCmd;
END_METHOD

METHOD PRIVATE _Scale : REAL
VAR_INPUT
    X    : REAL;
    I_LO : REAL;
    I_HI : REAL;
    O_LO : REAL;
    O_HI : REAL;
END_VAR
IF I_LO = I_HI THEN
	_Scale := O_LO;
ELSE
	_Scale := (O_HI - O_LO) / (I_HI - I_LO) * (LIMIT(I_LO, X, I_HI) - I_LO) + O_LO;
END_IF;
END_METHOD

END_FUNCTION_BLOCK

// ---- Function Blocks/PaperMachine/DriveControl/FB_FormingBoardControl_V3.TcPOU
FUNCTION_BLOCK FB_FormingBoardControl_V3

VAR_INPUT

    //────────────────────────────────────────────
    // GROUP / INTERLOCKS
    //────────────────────────────────────────────
    startGroup              : BOOL; // Start command (pulse) / Comando de partida (pulso)
    stopGroup               : BOOL; // Stop command (level) / Comando de parada (nível)
    fastStopGroup               : BOOL; // Stop command (level) / Comando de parada (nível)
	groupReset              : BOOL; // Fault reset / Reset de falhas do grupo
	
    //────────────────────────────────────────────
    // AUXILIARY MOTORS — INDICATORS & COMMANDS
    //────────────────────────────────────────────
    grouSpeedDifIncCmd      : BOOL; // Lamp: offset increasing / Lâmpada: aumento de offset
    grouSpeedDifDecCmd      : BOOL; // Lamp: offset decreasing / Lâmpada: redução de offset
	
    //────────────────────────────────────────────
    // SPEED ADJUSTMENTS / OFFSET TUNING
    //────────────────────────────────────────────
    groupRecoverSpeedCmd    : BOOL; // Recover speed while TRUE / Recuperar velocidade enquanto TRUE
    //────────────────────────────────────────────
    // DRIVE STATUS INPUTS — FORMING BOARD ROLLS
    //────────────────────────────────────────────
    tractionRollReady       : BOOL; // MASTER ready / Pronto (mestre)
    suctionRollReady        : BOOL; // SLAVE ready / Pronto (seguidor)
	paperPresenceSensor : BOOL;

    //────────────────────────────────────────────
    // SPEED SETPOINTS / MODE
    //────────────────────────────────────────────
    groupAutoSpeedMPM       : REAL;       // Auto mode speed [m/min]
    groupManualSpeedMPM     : REAL := 50.0; // Manual mode speed
    groupSpeedAutoMan       : BOOL;       // 0=Manual, 1=Auto

    //────────────────────────────────────────────
    // SPEED & TORQUE FEEDBACKS
    //────────────────────────────────────────────
    tractionRollSpeedFeedback     : REAL; // MASTER speed feedback
    tractionRollTorqueFeedback    : REAL; // MASTER torque feedback
    suctionRollSpeedFeedback      : REAL; // SLAVE speed feedback
    suctionRollTorqueFeedback     : REAL; // SLAVE torque feedback

    //────────────────────────────────────────────
    // WIRE/FELT EDGE / RUNNING SAFETY SENSORS
    //────────────────────────────────────────────
    formingBoardWireOverrunSensorOperatorSide : BOOL; // Operator side / Lado operador
    formingBoardWireOverrunSensorDriveSide    : BOOL; // Drive side / Lado comando

    machineConfig : PaperMachine_TypeHmiConfig;

END_VAR



VAR_OUTPUT

    //────────────────────────────────────────────
    // STATE / DIAGNOSTICS
    //────────────────────────────────────────────
    deviceState                 : STRING; // Current state string / Estado atual em texto
    statusCode                  : INT;    // 0=Idle, 1=Starting, 2=Running, 3=Fault
    groupFault                  : BOOL;   // TRUE if any group fault active / Falha geral do grupo
	speedDifError: BOOL;

    //────────────────────────────────────────────
    // SPEED REFERENCES (TO DRIVES) AND DISPLAY
    //────────────────────────────────────────────
    tractionRollSpeedSetpointRPM : REAL; // MASTER speed reference [rpm]
    suctionRollSpeedSetpointRPM  : REAL; // SLAVE speed reference [rpm]

    tractionRollSpeedFeedbackRPM : REAL; // MASTER speed feedback [rpm]
    suctionRollSpeedFeedbackRPM  : REAL; // SLAVE speed feedback [rpm]

    tractionRollSpeedFeedbackMPM : REAL; // MASTER speed feedback [m/min]
    suctionRollSpeedFeedbackMPM  : REAL; // SLAVE speed feedback [m/min]

    tractionRollTorqueFeedbackPct : REAL; // MASTER torque feedback [%]
    suctionRollTorqueFeedbackPct  : REAL; // SLAVE torque feedback [%]

    nextGroupSpeedRefMPM        : REAL; // Next group speed [m/min]

    //────────────────────────────────────────────
    // TORQUE REFERENCES / LIMITS (SLAVE)
    //────────────────────────────────────────────
    suctionRollTorqueRefPct     : REAL; // Torque setpoint for SLAVE [%]

    //────────────────────────────────────────────
    // DRIVE COMMANDS (ENABLE / RESET)
    //────────────────────────────────────────────
    tractionRollDriveEnable     : BOOL; // Enable MASTER drive
    tractionRollDriveReset      : BOOL; // Reset MASTER drive fault
    suctionRollDriveEnable      : BOOL; // Enable SLAVE drive
    suctionRollDriveReset       : BOOL; // Reset SLAVE drive fault

    //────────────────────────────────────────────
    // STATUS CODES (PER DRIVE)
    //────────────────────────────────────────────


    //────────────────────────────────────────────
    // HMI ALARMS STRUCTURE
    //────────────────────────────────────────────
    hmiAlarms                   : PaperMachine_TypeHmiAlarms;

END_VAR



VAR
    instFB_GroupDriveControl_V1       : FB_GroupDriveControl_V1;
    instFB_GroupSpeedControl_V1       : FB_GroupSpeedControl_V1;
	instFB_FormingBoardSpeedControl	: FB_FormingBoardSpeedControl;
    instFB_GroupDisplayFilters_V1     : FB_GroupDisplayFilters_V1;
    instFB_GroupTorqueTrimControl_V1  : FB_GroupTorqueTrimControl_V1;
	
	instFB_GroupTorqueTrimControl_V2  : FB_GroupTorqueTrimControl_V2;

	speedDif: REAL;
	instTONWireOverRunTrip: TON;
	instTONSpeedDifDelay: TON;
	instTOF_PaperPresenseDelay : TOF;	
	
	instTPSpeedDifErrorHold: TP;
END_VAR

VAR PERSISTENT
END_VAR

// ─────────────────────────────────────────────────────────────────────────────
// MAIN CALL SEQUENCE
// ─────────────────────────────────────────────────────────────────────────────

_GroupControl();          // 1) State machine: edges, enables, stop modes
_StateDisplay();
_SpeedDifferenceCheck();  // 4) Speed difference monitor & trip
_auxiliaryControls();

_alarmsDisplay();

METHOD _alarmsDisplay
VAR_INPUT
END_VAR
(*
//==============================================================
// FAULT EVALUATION — PER CONDITION (flags only; no global set)
//==============================================================

//----------------------------
// PRESS SECTION DRIVES
//----------------------------
hmiAlarms.pressSectionFirstPressFaultAlarm  := firstPressVfdFaultFeedback;
hmiAlarms.pressSectionSecondPressFaultAlarm := secondPressVfdFaultFeedback;

//----------------------------
// PRESS SECTION AUXILIARIES
//----------------------------
hmiAlarms.pressSectionUpperFeltStretcherFaultAlarm := upperFelt1StretcherFault;
hmiAlarms.pressSectionLowerFeltStretcherFaultAlarm := lowerFeltStretcherFault;
hmiAlarms.pressSectionUpperInfeedRollFaultAlarm    := upperInfeedRollFault;
hmiAlarms.pressSectionLowerInfeedRollFaultAlarm    := lowerInfeedRollFault;


//==============================================================
// PRESS SECTION — FELT EDGE OVERRUN ALARMS (DIRECT SENSORS)
//==============================================================

hmiAlarms.pressSectionUpperFelt1OverrunOperatorSideAlarm := pressSectionUpperFelt1OverrunSensorOperatorSide;
hmiAlarms.pressSectionUpperFelt1OverrunDriveSideAlarm    := pressSectionUpperFelt1OverrunSensorDriveSide;

hmiAlarms.pressSectionUpperFelt2OverrunOperatorSideAlarm := pressSectionUpperFelt2OverrunSensorOperatorSide;
hmiAlarms.pressSectionUpperFelt2OverrunDriveSideAlarm    := pressSectionUpperFelt2OverrunSensorDriveSide;

hmiAlarms.pressSectionLowerFeltOverrunOperatorSideAlarm := pressSectionLowerFeltOverrunSensorOperatorSide;
hmiAlarms.pressSectionLowerFeltOverrunDriveSideAlarm    := pressSectionLowerFeltOverrunSensorDriveSide;


//----------------------------
// PRESS SECTION GROUP FAULT STATUS
//----------------------------
groupFault :=
    hmiAlarms.pressSectionFirstPressFaultAlarm 
	OR hmiAlarms.pressSectionSecondPressFaultAlarm 
	OR hmiAlarms.pressFelt1OverrunOperatorSideAlarm
	OR hmiAlarms.pressFelt1OverrunDriveSideAlarm
	OR hmiAlarms.pressFelt2OverrunOperatorSideAlarm
	OR hmiAlarms.pressFelt2OverrunDriveSideAlarm
	OR hmiAlarms.pressFelt3OverrunOperatorSideAlarm
	OR hmiAlarms.pressFelt3OverrunDriveSideAlarm;


*)
//==============================================================
// FAULT EVALUATION — PER CONDITION (flags only; no global set)
//==============================================================

//----------------------------
// PRESS SECTION DRIVES
//----------------------------
//hmiAlarms.pressSectionFirstPressFaultAlarm  := firstPressVfdFaultFeedback;
//hmiAlarms.pressSectionSecondPressFaultAlarm := secondPressVfdFaultFeedback;

//----------------------------
// PRESS SECTION AUXILIARIES
//----------------------------
END_METHOD

METHOD _auxiliaryControls
VAR_INPUT
END_VAR
END_METHOD

METHOD _GroupControl
VAR_INPUT
END_VAR


(*
    formingBoardTorquePIDCtrlKp                   : REAL := 2.0;
    formingBoardTorquePIDCtrlTn                   : REAL := 8.0;
    formingBoardTorquePIDCtrlTv                   : REAL := 0.0;
    formingBoardTorqueLimit                   : REAL := 100.0;
	
*)
VAR
	suctionRollTorqueRefPct_: REAL;
END_VAR
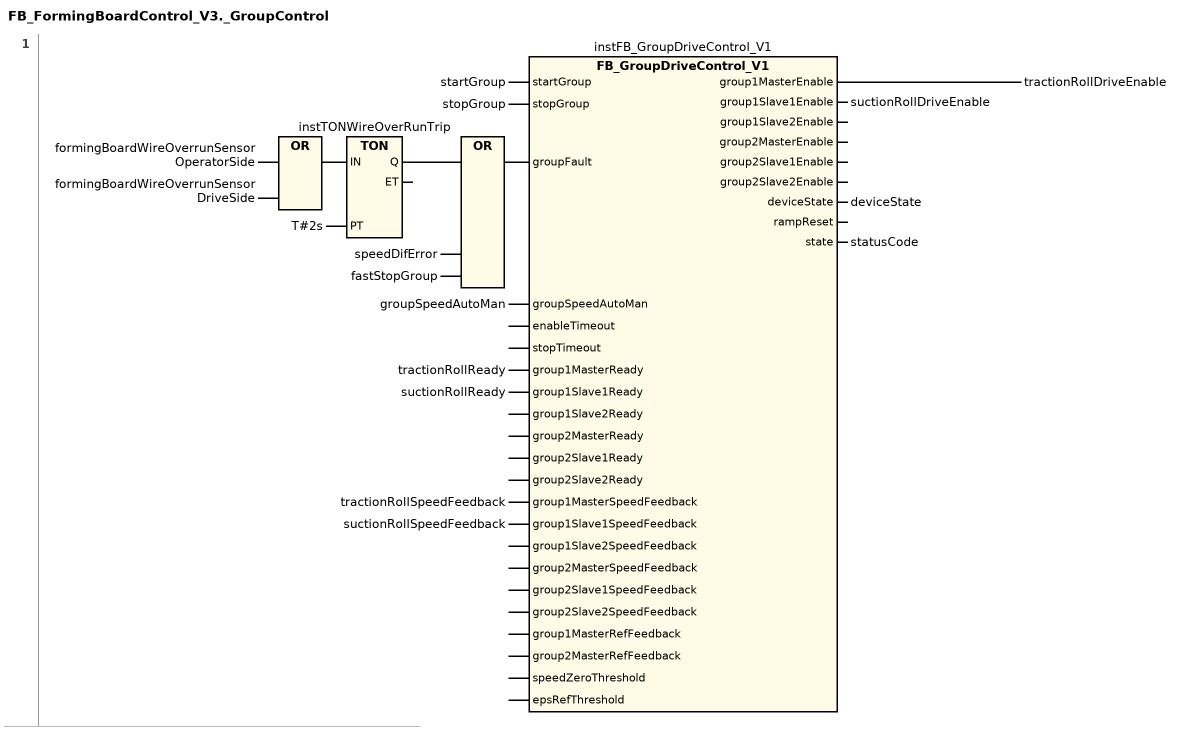
// NETWORK 1
instTONWireOverRunTrip(IN := formingBoardWireOverrunSensorOperatorSide OR formingBoardWireOverrunSensorDriveSide, PT := T#2s); // TON
instFB_GroupDriveControl_V1(
    startGroup := startGroup,
    stopGroup := stopGroup,
    groupFault := instTONWireOverRunTrip.Q OR speedDifError OR fastStopGroup,
    groupSpeedAutoMan := groupSpeedAutoMan,
    group1MasterReady := tractionRollReady,
    group1Slave1Ready := suctionRollReady,
    group1MasterSpeedFeedback := tractionRollSpeedFeedback,
    group1Slave1SpeedFeedback := suctionRollSpeedFeedback,
    group1Slave1Enable => suctionRollDriveEnable,
    deviceState => deviceState,
    state => statusCode); // FB_GroupDriveControl_V1
tractionRollDriveEnable := instFB_GroupDriveControl_V1.group1MasterEnable;

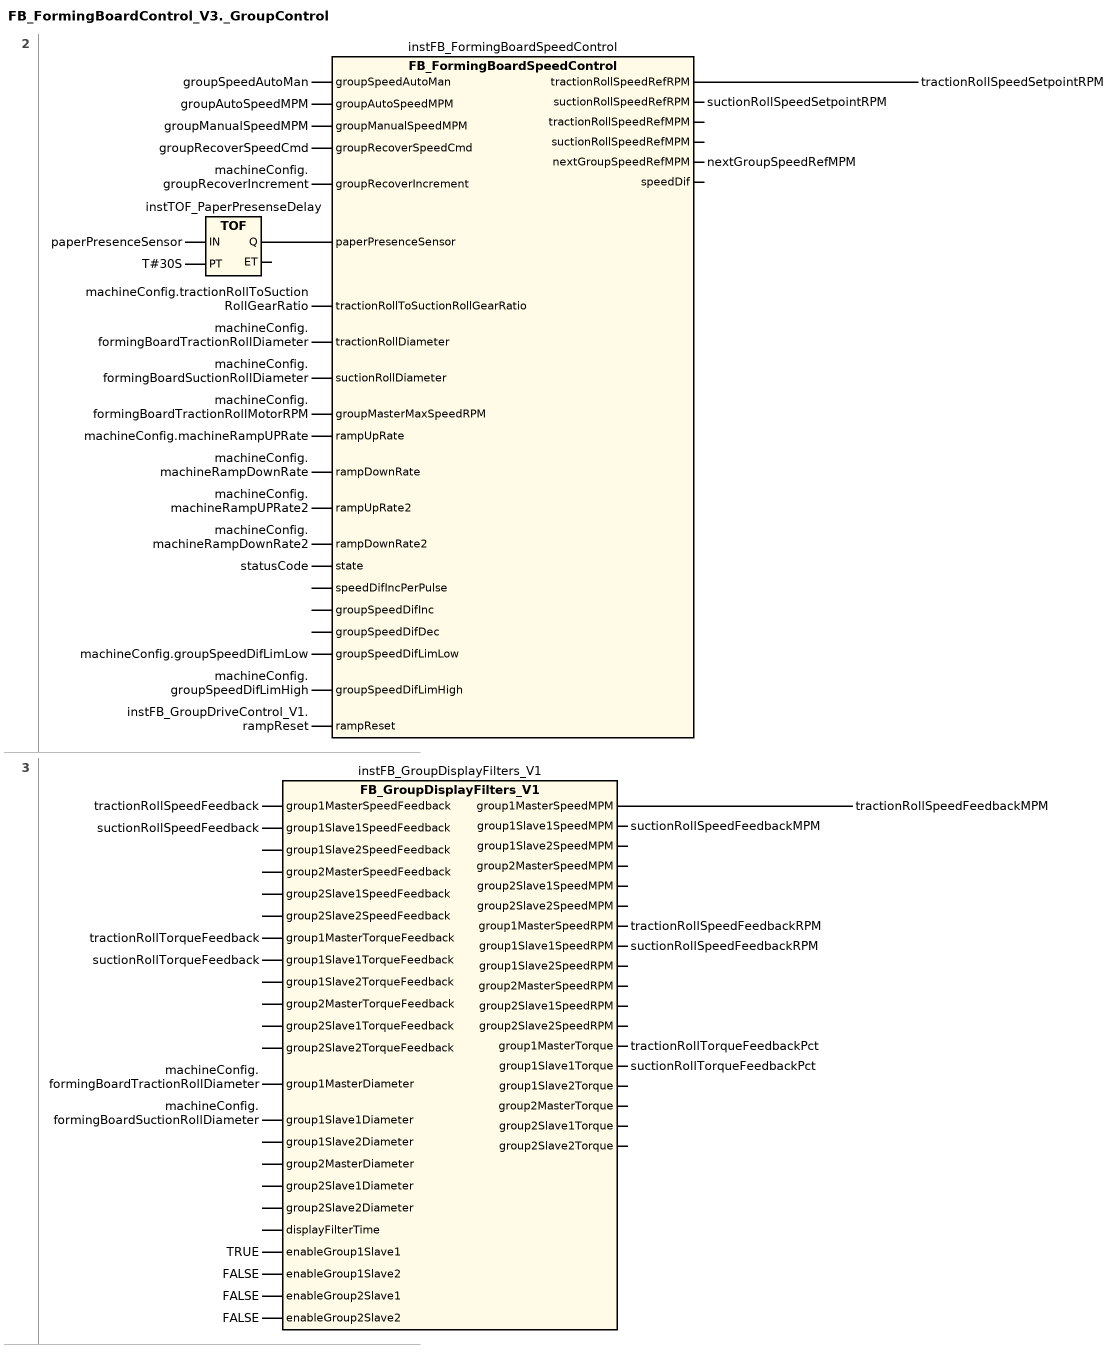
// NETWORK 2
instTOF_PaperPresenseDelay(IN := paperPresenceSensor, PT := T#30S); // TOF
instFB_FormingBoardSpeedControl(
    groupSpeedAutoMan := groupSpeedAutoMan,
    groupAutoSpeedMPM := groupAutoSpeedMPM,
    groupManualSpeedMPM := groupManualSpeedMPM,
    groupRecoverSpeedCmd := groupRecoverSpeedCmd,
    groupRecoverIncrement := machineConfig.groupRecoverIncrement,
    paperPresenceSensor := instTOF_PaperPresenseDelay.Q,
    tractionRollToSuctionRollGearRatio := machineConfig.tractionRollToSuctionRollGearRatio,
    tractionRollDiameter := machineConfig.formingBoardTractionRollDiameter,
    suctionRollDiameter := machineConfig.formingBoardSuctionRollDiameter,
    groupMasterMaxSpeedRPM := machineConfig.formingBoardTractionRollMotorRPM,
    rampUpRate := machineConfig.machineRampUPRate,
    rampDownRate := machineConfig.machineRampDownRate,
    rampUpRate2 := machineConfig.machineRampUPRate2,
    rampDownRate2 := machineConfig.machineRampDownRate2,
    state := statusCode,
    groupSpeedDifLimLow := machineConfig.groupSpeedDifLimLow,
    groupSpeedDifLimHigh := machineConfig.groupSpeedDifLimHigh,
    rampReset := instFB_GroupDriveControl_V1.rampReset,
    suctionRollSpeedRefRPM => suctionRollSpeedSetpointRPM,
    nextGroupSpeedRefMPM => nextGroupSpeedRefMPM); // FB_FormingBoardSpeedControl
tractionRollSpeedSetpointRPM := instFB_FormingBoardSpeedControl.tractionRollSpeedRefRPM;

// NETWORK 3
instFB_GroupDisplayFilters_V1(
    group1MasterSpeedFeedback := tractionRollSpeedFeedback,
    group1Slave1SpeedFeedback := suctionRollSpeedFeedback,
    group1MasterTorqueFeedback := tractionRollTorqueFeedback,
    group1Slave1TorqueFeedback := suctionRollTorqueFeedback,
    group1MasterDiameter := machineConfig.formingBoardTractionRollDiameter,
    group1Slave1Diameter := machineConfig.formingBoardSuctionRollDiameter,
    enableGroup1Slave1 := TRUE,
    enableGroup1Slave2 := FALSE,
    enableGroup2Slave1 := FALSE,
    enableGroup2Slave2 := FALSE,
    group1Slave1SpeedMPM => suctionRollSpeedFeedbackMPM,
    group1MasterSpeedRPM => tractionRollSpeedFeedbackRPM,
    group1Slave1SpeedRPM => suctionRollSpeedFeedbackRPM,
    group1MasterTorque => tractionRollTorqueFeedbackPct,
    group1Slave1Torque => suctionRollTorqueFeedbackPct); // FB_GroupDisplayFilters_V1
tractionRollSpeedFeedbackMPM := instFB_GroupDisplayFilters_V1.group1MasterSpeedMPM;

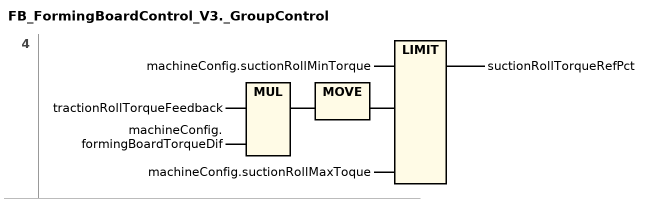
// NETWORK 4
suctionRollTorqueRefPct := LIMIT(machineConfig.suctionRollMinTorque, tractionRollTorqueFeedback * machineConfig.formingBoardTorqueDif, machineConfig.suctionRollMaxToque);
END_METHOD

METHOD PRIVATE _Scale : REAL
VAR_INPUT
    X    : REAL;
    I_LO : REAL;
    I_HI : REAL;
    O_LO : REAL;
    O_HI : REAL;
END_VAR
IF I_LO = I_HI THEN
	_Scale := O_LO;
ELSE
	_Scale := (O_HI - O_LO) / (I_HI - I_LO) * (LIMIT(I_LO, X, I_HI) - I_LO) + O_LO;
END_IF;
END_METHOD

// ============================== Methods ==============================
// Intra-section speed supervision for Press Section (firstPress ↔ secondPress)
METHOD _SpeedDifferenceCheck
(*

    tractionRollSpeedFeedbackMPM : REAL; // MASTER speed feedback [m/min]
    suctionRollSpeedFeedbackMPM  : REAL; // SLAVE speed feedback [m/min]

*)
speedDif := ABS(tractionRollSpeedFeedbackMPM - suctionRollSpeedFeedbackMPM);


// Timer de confirmação do erro
instTONSpeedDifDelay(
    IN := speedDif > 50,
    PT := T#3S
);


// Pulso para segurar o status do erro por 100 ms
instTPSpeedDifErrorHold(
    IN := instTONSpeedDifDelay.Q,
    PT := T#100MS
);


// Status final do erro
speedDifError := instTPSpeedDifErrorHold.Q;
END_METHOD

METHOD _StateDisplay
VAR_INPUT
END_VAR

// ──────────────────────────────────────────────────────────────────────────────
// _StateDisplay — Press Section (firstPress = Master, secondPress = Slave)
// Maps the internal machine "state" to a compact HMI status code and derives
// per-drive motor status codes from VFD signals.
//
// statusCode / firstPressStatusCode / secondPressStatusCode legend:
//   0 = Idle, 1 = Starting, 2 = Running, 3 = Fault
//
// Machine "state" groups:
//   0 = IDLE, 1 = ENABLE, 2 = WAIT_EN, 3 = RAMP_EN, 4 = RUN, 5 = STOPPING, 10 = FAULT
// Priority rule (for motors): Fault > Running > Starting > Idle
// ──────────────────────────────────────────────────────────────────────────────
VAR CONSTANT
    STATUS_IDLE     : INT := 0;
    STATUS_STARTING : INT := 1;
    STATUS_RUNNING  : INT := 2;
    STATUS_FAULT    : INT := 3;
END_VAR
END_METHOD

END_FUNCTION_BLOCK

// ---- Function Blocks/PaperMachine/FB_FormingBoardSpeedControl.TcPOU
FUNCTION_BLOCK FB_FormingBoardSpeedControl
VAR_INPUT
    //==============================================================
    // ─────────────── MODE SELECTION / REFERENCES ───────────────
    //==============================================================
    groupSpeedAutoMan          : BOOL;  // TRUE = Auto, FALSE = Manual
    groupAutoSpeedMPM          : REAL;  // Auto speed reference [m/min]
    groupManualSpeedMPM        : REAL;  // Manual speed reference [m/min]
    groupRecoverSpeedCmd       : BOOL;  // Recover (temporary speed bump)
    groupRecoverIncrement      : REAL;  // Recover increment [m/min]
//    interGroupGearRatio        : REAL;  // Inter-group ratio (next section sync)
	paperPresenceSensor				: BOOL;

    tractionRollToSuctionRollGearRatio  : REAL := 0.915;

    //==============================================================
    // ─────────────── DIAMETERS (mm) ───────────────
    //==============================================================
    tractionRollDiameter       : REAL;  // Diameter of group 1 master
    suctionRollDiameter       : REAL;  // Diameter of group 1 slave 1


    //==============================================================
    // ─────────────── CONFIGURATION / LIMITS ───────────────
    //==============================================================
    groupMasterMaxSpeedRPM     : REAL;  // Max allowed master RPM
    rampUpRate					: REAL := 0.1;  // Ramp slow acceleration [RPM/s]
    rampDownRate				: REAL := 0.1;  // Ramp slow acceleration [RPM/s]
	
    rampUpRate2					: REAL := 0.1;  // Ramp fast acceleration [RPM/s]
    rampDownRate2				: REAL := 0.1;  // Ramp fast acceleration [RPM/s]	
	
    state                      : INT;   // Machine state (5 = STOPPING)

	speedDifIncPerPulse		: REAL := 0.05;
	
    groupSpeedDifInc           : BOOL;  // Increment group speed offset
    groupSpeedDifDec           : BOOL;  // Decrement group speed offset
    groupSpeedDifLimLow        : REAL;  // Min offset [%]
    groupSpeedDifLimHigh       : REAL;  // Max offset [%]


    rampReset                  : BOOL;  // Reset ramp command
	
END_VAR


VAR_OUTPUT
    //==============================================================
    // ─────────────── FINAL DRIVE SPEEDS (RPM) ───────────────
    //==============================================================
    tractionRollSpeedRefRPM    : REAL; //Master speed
    suctionRollSpeedRefRPM    : REAL; // Slave speed

    //==============================================================
    // ─────────────── SURFACE SPEEDS (MPM) ───────────────
    //==============================================================
    tractionRollSpeedRefMPM       : REAL;
    suctionRollSpeedRefMPM       : REAL;


    //==============================================================
    // ─────────────── HANDOFF TO NEXT GROUP ───────────────
    //==============================================================
    nextGroupSpeedRefMPM       : REAL;
	speedDif					: REAL;
	
	
	
END_VAR


VAR
    //==============================================================
    // ─────────────── INTERNAL CALCULATION VARIABLES ───────────────
    //==============================================================
    masterMaxSpeedMPM          : REAL;
    baseCmdSpeedMPM            : REAL;
    cmdSpeedMPM                : REAL;
    targetRPM                  : REAL;
    rampTargetRPM              : REAL;
    baseMasterRefRPM           : REAL;
    groupSpeedOffset           : REAL;
    groupDeltaRatioAll         : REAL;
    upperLowerBiasRatio        : REAL;
    useRamp                    : BOOL;
    epsDiameter                : REAL := 0.001;

    // Gear ratios (set externally or calculated elsewhere)


    // Function blocks
    instFB_Gen_SRamp           : FB_Gen_SRamp;
    instFB_SpeedDif_SRamp           : FB_Gen_SRamp;

	rampActive: BOOL;
END_VAR


VAR PERSISTENT
	
    instTUNE2_GroupSpeedDiff   : TUNE2;

END_VAR

//==============================================================
// IMPLEMENTATION
//==============================================================

//====================================================================
// ═══ CALL METHOD TO CALCULATE DIAMETER RATIOS ═════════════════════
//====================================================================
_CalculateGearRatios();

//--------------------------------------------------------------
// Calculate master max surface speed [m/min]
//--------------------------------------------------------------
masterMaxSpeedMPM := groupMasterMaxSpeedRPM * (PI * tractionRollDiameter) / 1000.0;


//--------------------------------------------------------------
// Determine base speed source (auto/manual) + Recover bump
//--------------------------------------------------------------
IF groupSpeedAutoMan THEN
    baseCmdSpeedMPM := groupAutoSpeedMPM;
ELSE
    baseCmdSpeedMPM := groupManualSpeedMPM;
END_IF;

IF groupRecoverSpeedCmd THEN
    cmdSpeedMPM := baseCmdSpeedMPM + groupRecoverIncrement;
ELSE
    cmdSpeedMPM := baseCmdSpeedMPM;
END_IF;


//--------------------------------------------------------------
// Convert MPM → target RPM for the master
//--------------------------------------------------------------
targetRPM := _Scale(
    X    := cmdSpeedMPM,
    I_LO := 0.0,
    I_HI := masterMaxSpeedMPM,
    O_LO := 0.0,
    O_HI := groupMasterMaxSpeedRPM);


//--------------------------------------------------------------
// Ramp handling
//--------------------------------------------------------------
IF state = 5 OR state = 0 THEN
    // STOPPING — force ramp down to zero speed
    rampTargetRPM := 0.0;

ELSIF state = 10 THEN
    // FAULT — clear ramp immediately to ensure no residual motion
    rampTargetRPM := 0.0;
//    rampReset     := TRUE;

ELSE
    // Normal operation — ramp follows target speed
    rampTargetRPM := targetRPM;
//    rampReset     := FALSE;
END_IF;

// Detect when a new target speed change requires ramping
IF paperPresenceSensor THEN
 
  rampActive := TRUE; // Rising edge — ramp request detected

ELSE
	
  rampActive := FALSE; // Rising edge — ramp request detected
  
END_IF;



IF 	paperPresenceSensor THEN
	//slow	
	instFB_Gen_SRamp.A_UP := MAX(0.0, rampUpRate);
	instFB_Gen_SRamp.A_DN := -MAX(0.0, rampDownRate);

ELSE
	//fast
	instFB_Gen_SRamp.A_UP := MAX(0.0, rampUpRate2);
	instFB_Gen_SRamp.A_DN := -MAX(0.0, rampDownRate2);

END_IF


// Ramp function block execution
instFB_Gen_SRamp(
    X          := rampTargetRPM,
//    A_UP       := MAX(0.0, rampUpRate),
//    A_DN       := -MAX(0.0, rampDownRate),
    VU_MAX     := 1000.0,
    VD_MAX     := -1000.0,
    LIMIT_HIGH := groupMasterMaxSpeedRPM,
    RST        := rampReset);

// If ramping, update the baseMasterRefRPM from ramp output
IF rampActive THEN
    baseMasterRefRPM := instFB_Gen_SRamp.Y;

    // Automatically reset ramp flag when the ramp output reaches the target
    IF ABS(instFB_Gen_SRamp.Y - rampTargetRPM) <= 0.05 THEN
//        rampActive := FALSE; // Ramp complete
;
    END_IF;

ELSE
    // No ramping required — direct assignment
    baseMasterRefRPM := rampTargetRPM;
END_IF;


//--------------------------------------------------------------
// Operator offset (TUNE2 control)
//--------------------------------------------------------------
instTUNE2_GroupSpeedDiff(
    SET     := FALSE,
    SU      := groupSpeedDifInc,
    SD      := groupSpeedDifDec,
    RST     := FALSE,
    SS      := speedDifIncPerPulse,
    FS      := speedDifIncPerPulse,
    LIMIT_L := groupSpeedDifLimLow,
    LIMIT_H := groupSpeedDifLimHigh);
//    Y       => groupSpeedOffset);


// Ramp function block execution
instFB_SpeedDif_SRamp(
    X          := instTUNE2_GroupSpeedDiff.Y,
    A_UP       := MAX(0.0, 0.01),
    A_DN       := -MAX(0.0, 0.01),
    VU_MAX     := 1000.0,
    VD_MAX     := -1000.0,
    LIMIT_HIGH := groupSpeedDifLimHigh,
	LIMIT_LOW := groupSpeedDifLimLow,
    RST        := FALSE,
	Y => groupSpeedOffset);

	
speedDif := groupSpeedOffset;
	
groupDeltaRatioAll  := 1.0 + (groupSpeedOffset * 0.01);


//--------------------------------------------------------------
// Apply offsets + calculate all drive RPM references
//--------------------------------------------------------------
tractionRollSpeedRefRPM := baseMasterRefRPM * groupDeltaRatioAll;
suctionRollSpeedRefRPM := tractionRollSpeedRefRPM * tractionRollToSuctionRollGearRatio;


//--------------------------------------------------------------
// Convert RPM → MPM (surface speeds)
//--------------------------------------------------------------
tractionRollSpeedRefMPM := tractionRollSpeedRefRPM * tractionRollDiameter * PI / 1000.0;
suctionRollSpeedRefMPM := (suctionRollSpeedRefRPM * suctionRollDiameter * PI / 1000.0);



//--------------------------------------------------------------
// Suggest downstream handoff (group2 master surface speed)
//--------------------------------------------------------------
nextGroupSpeedRefMPM := tractionRollSpeedRefMPM;


//====================================================================
// ═══ PRIVATE METHOD — CALCULATE DIAMETER RATIOS ════════════════════
//====================================================================
METHOD PRIVATE _CalculateGearRatios
VAR_INPUT
END_VAR
END_METHOD

METHOD PRIVATE _Scale : REAL
VAR_INPUT
    X    : REAL;
    I_LO : REAL;
    I_HI : REAL;
    O_LO : REAL;
    O_HI : REAL;
END_VAR
IF I_LO = I_HI THEN
	_Scale := O_LO;
ELSE
	_Scale := (O_HI - O_LO) / (I_HI - I_LO) * (LIMIT(I_LO, X, I_HI) - I_LO) + O_LO;
END_IF;
END_METHOD

END_FUNCTION_BLOCK

// ---- Function Blocks/PaperMachine/Auxiliary/FB_SimpleMotorStart_V3.TcPOU
FUNCTION_BLOCK FB_SimpleMotorStart_V3
VAR_INPUT
    // ───────── Commands & interlocks ─────────
    startCommand                 : BOOL;   // Pulse to toggle run (Pulso para alternar execução)
    stopCommand                  : BOOL;   // Pulse to force stop (Pulso para forçar parada
	runtimeMeterResetCmd		: BOOL;
	
    motorStarterOK             : BOOL := TRUE;   // Softstarter healthy/ready (Softstarter ok/pronto)
    safetyOK                   	 : BOOL	:= TRUE;   // External interlock 1 (Intertravamento 1)
	
    interlock1                   : BOOL := TRUE;   // External interlock 2 (Intertravamento 2)
    interlock2                   : BOOL := TRUE;   // External interlock 3 (Intertravamento 3)
    interlock3                   : BOOL := TRUE;   // External interlock 4 (Intertravamento 4)

    // ───────── Motor current proof ─────────
    motorCurrentFeedback         : REAL;   // Measured motor current

END_VAR

VAR_OUTPUT
	
    faultActive                  : BOOL;       // Latched fault
	lineContactor                : BOOL;       // CMD line/bypass contactor
    deviceState                  : STRING(80); // Human-readable state
    statusCode                   : INT;        // 0=Idle, 1=Running, 2=Fault
    motorCurrentFiltered         : REAL;       // Filtered motor current for HMI/logic
	runtimeMeter				 : DINT;
	
END_VAR

VAR
    // ───────── State & edges ─────────
    step                         : INT;    // State machine step
    startCommandOld              : BOOL;
    stopCommandOld               : BOOL;
    rStart                       : BOOL;
    rStop                        : BOOL;

    // ───────── Latch ─────────
    runLatch                     : BOOL;   // Latched run request (start toggles, stop clears)

    // ───────── Timers ─────────
    tonStartDelay                : TON;    // Ramp-up timer

    // ───────── Helpers ─────────
    allInterlocksOK              : BOOL;
    proofCurrent                 : REAL;

    // ───────── OSCAT PT1 instance used by _InputFilter ─────────
    // Replace FT_PT1T with the correct type name from your OSCAT lib if different.
    instsFT_PT1TInputFilter      : FT_PT1;

END_VAR

// ============================ Edges, interlocks, defaults ============================
rStart := startCommand AND NOT startCommandOld;
rStop  := stopCommand  AND NOT stopCommandOld;
startCommandOld := startCommand;
stopCommandOld  := stopCommand;

allInterlocksOK := safetyOK AND interlock1 AND interlock2 AND interlock3;

// Start TOGGLES run latch; Stop forces stop
IF rStart THEN
    runLatch := NOT runLatch;  // Toggle / Alterna start-stop
END_IF;

IF rStop THEN
    runLatch := FALSE;         // Stop sempre desliga
END_IF;

// Default textual state
deviceState := 'Idle (Parado)';

// =============================== Fault reset =======================================
// Limpa falha somente quando não há pedido de partida e stop não está mantido
IF NOT runLatch AND NOT stopCommand THEN
    faultActive := FALSE;
END_IF;

// ============================= Interlocks & health checks ===========================
// Se pedir para rodar sem intertravamento ou softstarter OK -> entra em falha
IF runLatch AND NOT allInterlocksOK THEN
    faultActive := TRUE;
    deviceState := 'Fault: interlock open (Falha: intertrav. aberto)';
END_IF;

IF runLatch AND NOT motorStarterOK THEN
    faultActive := TRUE;
    deviceState := 'Fault: softstarter not OK (Falha: softstarter NOK)';
END_IF;

// Se falha ativa, garante tudo parado e volta pro passo 0
IF faultActive THEN
    lineContactor := FALSE;
    step := 0;
END_IF;

// ============================= Stop handling (immediate) ===========================
// Stop (pulso ou nível) força parada imediata
IF rStop OR stopCommand THEN
    lineContactor := FALSE;
    tonStartDelay(IN := FALSE);
    runLatch := FALSE;       // garante que o latch desligue
    step := 0;
END_IF;

// ================================= State machine ===================================
// Máquina de estados simples: 0 = Idle, 10 = Starting delay, 50 = Running
CASE step OF

    // ---------------------------------------------------------
    // 0: IDLE
    // ---------------------------------------------------------
    0:
        lineContactor := FALSE;
        tonStartDelay(IN := FALSE);
        deviceState := 'Idle (Parado)';

        // Condições para iniciar partida
        IF runLatch AND NOT faultActive AND motorStarterOK AND allInterlocksOK AND NOT stopCommand THEN
            // Inicia tempo de partida (ajuste o PT conforme desejado)
            tonStartDelay(IN := TRUE, PT := T#10MS);
            deviceState := 'Starting (Partida - softstarter)';
            step := 10;
        END_IF;


    // ---------------------------------------------------------
    // 10: STARTING DELAY (SOFTSTARTER)
    // ---------------------------------------------------------
    10:
        deviceState := 'Starting (Partida - softstarter)';
        tonStartDelay(IN := TRUE, PT := T#10MS);

        // Abort start se perder condição
        IF NOT runLatch OR stopCommand OR faultActive OR NOT allInterlocksOK OR NOT motorStarterOK THEN
            tonStartDelay(IN := FALSE);
            lineContactor := FALSE;
            step := 0;

        ELSIF tonStartDelay.Q THEN
            // Tempo de partida concluído -> liga contator de linha
            tonStartDelay(IN := FALSE);
            lineContactor := TRUE;
            step := 50;
        END_IF;


    // ---------------------------------------------------------
    // 50: RUNNING ON LINE
    // ---------------------------------------------------------
    50:
        lineContactor := TRUE;
        deviceState := 'Running on line (Operando em linha)';

        // Sai do RUN se o latch for desligado ou se der stop
        IF NOT runLatch OR stopCommand THEN
            lineContactor := FALSE;
            step := 0;
        END_IF;


    // ---------------------------------------------------------
    // Fallback (qualquer outro valor de step)
    // ---------------------------------------------------------
    ELSE
        lineContactor := FALSE;
        tonStartDelay(IN := FALSE);
        deviceState := 'Idle (Parado)';
        step := 0;
END_CASE;


// =============================== Status code =======================================
// 0 = Idle/Off
// 1 = Running
// 2 = Fault
IF faultActive THEN
    statusCode := 2;             // Fault
ELSIF lineContactor THEN
    statusCode := 1;             // Running
ELSE
    statusCode := 0;             // Idle / Off
END_IF;

// ============================================================================
// METHOD: _InputFilter
// OSCAT PT1 filter for PV, with enable/disable and bumpless behavior.
// When disabled, the filter tracks input quickly (tiny T) to avoid bumps.
// ============================================================================
METHOD PRIVATE _InputFilter
VAR_INPUT
    enableFilter   : BOOL;  // TRUE=apply PT1, FALSE=bypass
    rawValue       : REAL;  // Input value to be filtered
    filterTime     : TIME;  // PT1 time constant
    filterGainK    : REAL;  // PT1 gain, typically 1.0
END_VAR
VAR_OUTPUT
    filteredValue  : REAL;  // Filtered (or bypassed) value
END_VAR
VAR
    kUse           : REAL;
    tUse           : TIME;
    yPT1           : REAL;
END_VAR


IF enableFilter THEN
    kUse := filterGainK;
    tUse := filterTime;
ELSE
    // Track input closely for bumpless re-enable
    kUse := 1.0;
    tUse := T#10ms;
END_IF;

instsFT_PT1TInputFilter(
    in  := rawValue,
    T   := tUse,
    K   := kUse,
    out => yPT1
);

// Output selection
IF enableFilter THEN
    filteredValue := yPT1;
ELSE
    filteredValue := rawValue;
END_IF;
END_METHOD

END_FUNCTION_BLOCK

// ---- Function Blocks/PaperMachine/Auxiliary/FB_JumboWeightCapture.TcPOU
FUNCTION_BLOCK FB_JumboWeightCapture
VAR_INPUT
    currentWeightKg        : REAL;              // Live weight continuously supplied by the HMI
    shaftSelector          : INT;               // Selected shaft index, from 1 through 20
    shaftWeightKg          : ARRAY[1..20] OF REAL; // Persistent shaft tare weights [kg]
    captureRequest         : BOOL;              // Capture on rising edge only
    minimumCaptureInterval : TIME := T#10S;     // Protection against accidental repeated captures
END_VAR

VAR_OUTPUT
    capturedWeightKg       : REAL;              // Last accepted net weight [kg]
    capturedShaftSelector  : INT;               // Shaft selector latched with the accepted capture
    capturedAtFileTime     : ULINT;             // UTC Windows FILETIME, 100 ns ticks since 1601-01-01
    captureEventCounter    : UDINT;             // Monotonic event discriminator during PLC runtime
    captureReady           : BOOL;              // TRUE when a new rising edge can be accepted
    captureStatus          : INT;               // Stable operator status code for HMI text mapping
END_VAR

VAR
    initialized            : BOOL;
    captureRequestOld      : BOOL;
    captureRequestRising   : BOOL;
    captureInhibitActive   : BOOL;
    captureInhibitTimer    : TON;
    captureAcceptedPulse   : BOOL;
    captureBlockedPulse    : BOOL;
    captureSuccessTimer    : TP;
    captureBlockedTimer    : TP;
    shaftSelectorValid     : BOOL;
    shaftWeightValid       : BOOL;
    netWeightValid         : BOOL;
    selectedShaftWeightKg  : REAL;
END_VAR

VAR CONSTANT
    STATUS_INITIALIZING          : INT := 0;
    STATUS_READY                 : INT := 10;
    STATUS_CAPTURED              : INT := 20;
    STATUS_WAITING_INTERVAL      : INT := 30;
    STATUS_REQUEST_BLOCKED       : INT := 40;
    STATUS_RELEASE_REQUEST       : INT := 50;
    STATUS_INVALID_SHAFT         : INT := 60;
    STATUS_SHAFT_NOT_CONFIGURED  : INT := 70;
    STATUS_INVALID_NET_WEIGHT    : INT := 80;
END_VAR

// Initialize the edge memory from the actual input. This avoids an unintended
// capture when the PLC starts while the HMI request is already TRUE.
IF NOT initialized THEN
    captureRequestOld := captureRequest;
    initialized := TRUE;
    captureReady := FALSE;
    captureStatus := STATUS_INITIALIZING;
    RETURN;
END_IF

captureRequestRising := captureRequest AND NOT captureRequestOld;
captureAcceptedPulse := FALSE;
captureBlockedPulse := FALSE;

// Resolve the selected tare only after validating the array index. A zero or
// negative tare is treated as an unconfigured shaft.
shaftSelectorValid := shaftSelector >= 1 AND shaftSelector <= 20;
IF shaftSelectorValid THEN
    selectedShaftWeightKg := shaftWeightKg[shaftSelector];
ELSE
    selectedShaftWeightKg := 0.0;
END_IF

shaftWeightValid := shaftSelectorValid AND selectedShaftWeightKg > 0.0;
netWeightValid := shaftWeightValid AND currentWeightKg > selectedShaftWeightKg;

// The timer blocks accidental double captures. Reset it explicitly after Q so
// that a capture accepted on the expiry cycle starts a complete new interval.
captureInhibitTimer(
    IN := captureInhibitActive,
    PT := minimumCaptureInterval
);

IF captureInhibitTimer.Q THEN
    captureInhibitActive := FALSE;
    captureInhibitTimer(
        IN := FALSE,
        PT := minimumCaptureInterval
    );
END_IF

IF captureRequestRising AND NOT captureInhibitActive AND netWeightValid THEN
    capturedWeightKg := currentWeightKg - selectedShaftWeightKg;
    capturedShaftSelector := shaftSelector;
    capturedAtFileTime := F_GetSystemTime();
    captureEventCounter := captureEventCounter + 1;
    captureInhibitActive := minimumCaptureInterval > T#0S;
    captureAcceptedPulse := TRUE;
ELSIF captureRequestRising AND captureInhibitActive THEN
    captureBlockedPulse := TRUE;
END_IF

// Short, deterministic feedback windows make success and rejection visible
// even when the HMI button is only pulsed for one PLC cycle.
captureSuccessTimer(
    IN := captureAcceptedPulse,
    PT := T#2S
);
captureBlockedTimer(
    IN := captureBlockedPulse,
    PT := T#2S
);

// A new capture requires both the protection interval to have elapsed and the
// HMI request to be released, so the next command always creates a new edge.
captureReady := NOT captureInhibitActive AND NOT captureRequest AND netWeightValid;

IF captureBlockedTimer.Q THEN
    captureStatus := STATUS_REQUEST_BLOCKED;
ELSIF captureSuccessTimer.Q THEN
    captureStatus := STATUS_CAPTURED;
ELSIF NOT shaftSelectorValid THEN
    captureStatus := STATUS_INVALID_SHAFT;
ELSIF NOT shaftWeightValid THEN
    captureStatus := STATUS_SHAFT_NOT_CONFIGURED;
ELSIF NOT netWeightValid THEN
    captureStatus := STATUS_INVALID_NET_WEIGHT;
ELSIF captureRequest THEN
    captureStatus := STATUS_RELEASE_REQUEST;
ELSIF captureInhibitActive THEN
    captureStatus := STATUS_WAITING_INTERVAL;
ELSE
    captureStatus := STATUS_READY;
END_IF

captureRequestOld := captureRequest;

END_FUNCTION_BLOCK

// ---- Function Blocks/PaperMachine/Auxiliary/FB_WirePitControl_1.TcPOU
(*
    FB_ProcessControler
    Purpose: Generic process controller with start/stop latch, status codes,
             PID (OSCAT CTRL_PID), optional reverse action, PV PT1 filter,
             engineering↔% scaling, drive run supervision, and HMI displays.

    Sequence: Start pulse toggles RUN latch; Stop pulse/level forces stop.

    Status codes: statusCode INT → 0=Idle, 1=Running, 2=Fault

    Notes: Includes optional low/high PV “hold” with hysteresis (normal-stop class).
*)

FUNCTION_BLOCK FB_WirePitControl_1
VAR_INPUT
    // ===== Sequence commands =====
    startCommand                 : BOOL;            // Start pulse toggles RUN latch
    stopCommand                  : BOOL;            // Stop pulse/level forces stop

    // ===== Manual output & Auto SP nudge =====
    processSetpointManInc        : BOOL;            // Manual output ↑ (0..100%)
    processSetpointManDec        : BOOL;            // Manual output ↓ (0..100%)
    processSetpointManSteps      : REAL := 0.1;

    processSetpointAutoInc       : BOOL;            // Auto SP ↑ (engineering units or %)
    processSetpointAutoDec       : BOOL;            // Auto SP ↓ (engineering units or %)
    processSetpointAutoSteps     : REAL := 1.0;

    // ===== Mode =====
    autoMode                     : BOOL;            // TRUE=Automatic / FALSE=Manual
    reverseActing                : BOOL := FALSE;   // TRUE: higher output decreases PV; FALSE: direct

    // ===== Process signals (PV in engineering units) =====
    wirePitLevel           : REAL;            // PV (engineering units), e.g., bar/kPa/°C/…
	whiteWaterSiloLevel			: REAL;
    // ===== PID parameters (OSCAT CTRL_PID) =====
    kp                           : REAL := 1.0;     // Proportional gain (sign handled via reverseActing)
    tn                           : REAL := 8.0;     // Integral time [s]
    tv                           : REAL := 0.0;     // Derivative time [s]

    // ===== Output limits & offset =====
    outLowLimitPct               : REAL := 0.0;     // Min output %
    outHighLimitPct              : REAL := 100.0;   // Max output %
    outputOffsetPct              : REAL := 0.0;     // Offset added to final output

    // ===== PID housekeeping =====
    resetPID                     : BOOL;            // Reset integrator

    // ===== Input filter (OSCAT FT_PT1) =====
    enableInputFilter            : BOOL := TRUE;    // Enable PV PT1 filter
    inputFilterTime              : TIME := T#300ms; // PT1 time constant
    inputFilterGainK             : REAL := 1.0;     // PT1 gain

    displayFilterTime            : TIME := T#20ms;  // Small PT1 for HMI displays

    // ===== Optional scaling (engineering ↔ %) =====
    enableScaling                : BOOL := TRUE;    // Enable engineering↔% scaling
    pLoEng                       : REAL := 0.0;     // Engineering low bound
    pHiEng                       : REAL := 10.0;    // Engineering high bound

    // ===== Drive interface & supervision (VFD or actuator drive) =====
    vfdReady                     : BOOL;            // Drive ready/healthy
    vfdRunFeedback               : BOOL;            // Drive RUN feedback
    vfdFaultFeedback             : BOOL;            // Drive fault
    vfdRunFbTimeout              : TIME := T#5s;    // Timeout to receive RUN FB after start

    // ===== Drive analog feedbacks (for HMI display) =====
    vfdCurrentFeedback           : REAL;            // Current [A or %]
    vfdEngFeedback               : REAL;            // Engineering feedback (e.g., rpm, flow, etc.)
    vfdTorqueFeedback            : REAL;            // Torque (Nm or %)

    // ===== Safety (true safety inputs only) =====
    safetyOk                     : BOOL := TRUE;    // Safety chain OK
    estopOk                      : BOOL := TRUE;    // E-Stop loop OK
    guardClosedOk                : BOOL := TRUE;    // Guards/doors closed

    // ===== Interlocks (process permissives) — normal stop only =====
    interlock1                   : BOOL := TRUE;
    interlock2                   : BOOL := TRUE;
    interlock3                   : BOOL := TRUE;
    interlock4                   : BOOL := TRUE;
    interlock5                   : BOOL := TRUE;
    interlock6                   : BOOL := TRUE;

 // ===== Optional low-PV hold (normal-stop/hold) =====
    minPVEnable                  : BOOL := FALSE;   // Enable low-PV hold
    minPVTripEng                 : REAL := 0.5;     // Trip threshold (engineering units)
    minPVReleaseEng              : REAL := 0.7;     // Release threshold (engineering units)
    minPVTripTime                : TIME := T#1s;    // PV < trip for this long to trip
    minPVReleaseTime             : TIME := T#1s;    // PV > release for this long to release

    // ===== Optional high-PV hold (normal-stop/hold) =====
    maxPVEnable                  : BOOL := FALSE;   // Enable high-PV hold
    maxPVTripEng                 : REAL := 9.5;     // Trip threshold (engineering units)
    maxPVReleaseEng              : REAL := 9.2;     // Release threshold (engineering units)
    maxPVTripTime                : TIME := T#1s;    // PV > trip for this long to trip
    maxPVReleaseTime             : TIME := T#1s;    // PV < release for this long to release
	
	
END_VAR

VAR_OUTPUT
    running                      : BOOL;            // TRUE only during RUN state
    controlOutputPct             : REAL;            // Final control output 0..100%
    pidDiff                      : REAL;            // SET − ACT (post-scaling)
    pidLimited                   : BOOL;            // TRUE if saturated
    deviceState                  : STRING(80);      // Human-readable state
    vfdStartCmdOut               : BOOL;            // Asserted in Start/Run to the drive

    // ===== Holds (normal stop class) =====
    minPressureHoldActive        : BOOL;            // Low-PV hold active
    maxPressureHoldActive        : BOOL;            // High-PV hold active

    // ===== Status & HMI displays =====
    statusCode                   : INT;             // 0=Idle, 1=Running, 2=Fault
    vfdCurrentDisplay            : REAL;            // Display current [A or %]
    vfdTorqueDisplay             : REAL;            // Display torque (Nm or %)
    vfdEngDisplay                : REAL;            // Display engineering feedback (e.g., rpm)
    wirePitLevelDisplay    : REAL;            // PV (engineering units), e.g., bar/kPa/°C/…
	whiteWaterSiloLevelDisplay		: REAL;
	
END_VAR

VAR
    // ===== First scan & state/edges =====
    firstScan                    : BOOL := TRUE;    // TRUE only on first PLC cycle
	pvHoldActive 				 : BOOL;
    step                         : INT;             // 0=Idle,10=Starting,20=Running,90=Stopping
    startOld                     : BOOL;            // Edge memory
    stopOld                      : BOOL;            // Edge memory
    rStart                       : BOOL;            // Rising edge: start
    rStop                        : BOOL;            // Rising edge: stop
    runLatch                     : BOOL;            // Toggled by Start; cleared by Stop

    // ===== Internals =====
    manualCmd                    : REAL;            // Manual command %
    yPID                         : REAL;            // PID output %
    kpUse                        : REAL;            // Kp adjusted by reverseActing

    // ===== Filtered PV (engineering units) =====
    pvEngFiltered                : REAL;

    // ===== PV & SP in % (post-scaling) =====
    pvPct                        : REAL;
    spPct                        : REAL;

    // ===== Timers =====
    tonRunFbWait                 : TON;             // Waits RUN FB after start

    // ===== Low/High PV timers =====
    tonMinPTrip                  : TON;
    tonMinPRelease               : TON;
    tonMaxPTrip                  : TON;
    tonMaxPRelease               : TON;

    // ===== Instances =====
    instPID                      : CTRL_PID;        // OSCAT PID
    instPT1                      : FT_PT1;          // PV PT1 filter

    // ===== Aggregations =====
    allSafetyOK                  : BOOL;            // safetyOk & estopOk & guardClosedOk
    anyInterlockOpen             : BOOL;            // any interlock is FALSE

    // ===== HMI display filters =====
    instPT1_TorqueDisplay        : FT_PT1;          // PT1 for torque display
    instPT1_SpeedDisplay         : FT_PT1;          // PT1 for engineering display
	
    instPT1_ProcessFeedbackEngDisplay        : FT_PT1;          // PT1 for engineering display
	instPT1_WhiteWaterSiloLevelDisplay        : FT_PT1;          // PT1 for engineering display


    processSetpointManOld        : REAL;            // Last observed manual SP (HMI)
    processSetpointAutoOld       : REAL;            // Last observed auto SP (HMI)
	minPVHoldActive: BOOL;
	maxPVHoldActive: BOOL;
END_VAR

VAR PERSISTENT
    instTUNE2AutoSetpoint        : TUNE2;           // OSCAT TUNE2 for auto SP nudge
    instTUNE2ManSetpoint         : TUNE2;           // OSCAT TUNE2 for manual output
END_VAR

VAR_IN_OUT
    // ===== Exposed setpoints =====
    processSetpointMan           : REAL;            // Manual output 0..100%
    processSetpointAuto          : REAL;            // Auto SP (engineering units or % per configuration)
END_VAR

// ============================ INITIALIZATION ============================
// Run this block only once on first cycle
IF firstScan THEN
    firstScan := FALSE;

    processSetpointMan      := instTUNE2ManSetpoint.Y;
    processSetpointManOld   := processSetpointMan;

    processSetpointAuto     := instTUNE2AutoSetpoint.Y;
    processSetpointAutoOld  := processSetpointAuto;
END_IF;


// ============================ Edges ============================
rStart := startCommand AND NOT startOld;
startOld := startCommand;

rStop  := stopCommand AND NOT stopOld;
stopOld := stopCommand;

// Start toggles run; Stop forces stop
IF rStart THEN
    runLatch := TRUE;
END_IF;
IF rStop OR stopCommand THEN
    runLatch := FALSE;
END_IF;


// ============================ Aggregations =====================
allSafetyOK := safetyOk AND estopOk AND guardClosedOk;
anyInterlockOpen := NOT (interlock1 AND interlock2 AND interlock3 AND interlock4 AND interlock5 AND interlock6);

// Defaults each cycle
vfdStartCmdOut := FALSE;


// ============================ Low/High PV HOLD supervision ============================
// LOW-PV - Hold if the wire pit level is too low
IF minPVEnable AND autoMode THEN
    tonMinPTrip   (IN := (wirePitLevel <  minPVTripEng),     PT := minPVTripTime);
    tonMinPRelease(IN := (wirePitLevel >  minPVReleaseEng),  PT := minPVReleaseTime);
    IF tonMinPTrip.Q    THEN minPVHoldActive := TRUE;  END_IF;
    IF tonMinPRelease.Q THEN minPVHoldActive := FALSE; END_IF;

ELSE
    tonMinPTrip(IN := FALSE);
    tonMinPRelease(IN := FALSE);
    minPVHoldActive := FALSE;
END_IF;

// HIGH-PV - Hold if the silo level is too high
IF maxPVEnable AND autoMode THEN
    tonMaxPTrip   (IN := (whiteWaterSiloLevel > maxPVTripEng),       PT := maxPVTripTime);
    tonMaxPRelease(IN := (whiteWaterSiloLevel < maxPVReleaseEng),    PT := maxPVReleaseTime);
    IF tonMaxPTrip.Q    THEN maxPVHoldActive := TRUE;  END_IF;
    IF tonMaxPRelease.Q THEN maxPVHoldActive := FALSE; END_IF;

ELSE
    tonMaxPTrip(IN := FALSE);
    tonMaxPRelease(IN := FALSE);
    maxPVHoldActive := FALSE;
END_IF;

// ============================ PV HOLD aggregation ============================
// NOTE: Requires pvHoldActive : BOOL in VAR section
pvHoldActive := FALSE;
IF autoMode THEN
    pvHoldActive := (minPVEnable AND minPVHoldActive) OR
                    (maxPVEnable AND maxPVHoldActive);
END_IF;


// ============================ Immediate stop / safety/fault =================
IF rStop OR stopCommand THEN
    controlOutputPct := 0.0;
    running := FALSE;
    deviceState := 'Stopping (Stop command)';
    runLatch := FALSE;
    step := 90;
END_IF;

IF vfdFaultFeedback THEN
    deviceState := 'Fault from drive';
    runLatch := FALSE;
    step := 90;
END_IF;

IF NOT allSafetyOK THEN
    deviceState := 'Stopping: safety chain open';
    runLatch := FALSE;
    step := 90;
END_IF;


// ============================ State machine =====================
CASE step OF
    // ------------------------------------------------------------
    0: // Idle
        running := FALSE;
        controlOutputPct := 0.0;
        deviceState := 'Idle';
        vfdStartCmdOut := FALSE;

        // Start request via runLatch (toggled by Start pulse)
        IF runLatch AND NOT stopCommand THEN
            // Safety must be OK; drive must be ready
            // PV hold does NOT block start anymore; it will only inhibit reference to 0%
            IF NOT allSafetyOK THEN
                deviceState := 'Start blocked: safety not OK';
                runLatch := FALSE;
                step := 0;

            ELSIF NOT vfdReady THEN
                deviceState := 'Start blocked: drive not ready';
                runLatch := FALSE;
                step := 0;

            ELSE
                IF pvHoldActive THEN
                    deviceState := 'Starting (PV hold active: output inhibited)';
                ELSE
                    deviceState := 'Starting';
                END_IF;

                vfdStartCmdOut := TRUE;                   // send START to drive
                tonRunFbWait(IN := TRUE, PT := vfdRunFbTimeout);
                step := 10;
            END_IF
        END_IF

    // ------------------------------------------------------------
    10: // Starting (await RUN feedback)
        running := FALSE;
        deviceState := 'Starting (await RUN feedback)';
        vfdStartCmdOut := TRUE;

        // If PV hold is active during start, ensure reference is inhibited to 0%
        IF pvHoldActive THEN
            controlOutputPct := 0.0;
        END_IF;

        // Safety/fault during start => stop
        IF NOT allSafetyOK THEN
            tonRunFbWait(IN := FALSE);
            deviceState := 'Stopping: safety chain open';
            vfdStartCmdOut := FALSE;
            runLatch := FALSE;
            step := 90;

        ELSIF vfdFaultFeedback THEN
            tonRunFbWait(IN := FALSE);
            deviceState := 'Fault from drive';
            vfdStartCmdOut := FALSE;
            runLatch := FALSE;
            step := 90;

        // Interlocks are normal stop only
        ELSIF anyInterlockOpen THEN
            tonRunFbWait(IN := FALSE);
            deviceState := 'Stopping: interlock open';
            vfdStartCmdOut := FALSE;
            runLatch := FALSE;
            step := 90;

        // RUN feedback arrived
        ELSIF vfdRunFeedback THEN
            tonRunFbWait(IN := FALSE);
            step := 20;

        // Timeout
        ELSIF tonRunFbWait.Q THEN
            tonRunFbWait(IN := FALSE);
            deviceState := 'Start failed: RUN feedback timeout';
            vfdStartCmdOut := FALSE;
            runLatch := FALSE;
            step := 90;
        END_IF

    // ------------------------------------------------------------
    20: // Running (control loop)
        running := TRUE;               // may be used to release other devices
        deviceState := 'Running';
        vfdStartCmdOut := TRUE;

        // Supervision
        IF NOT allSafetyOK THEN
            deviceState := 'Stopping: safety chain open';
            vfdStartCmdOut := FALSE;
            runLatch := FALSE;
            step := 90;

        ELSIF vfdFaultFeedback THEN
            deviceState := 'Fault from drive';
            vfdStartCmdOut := FALSE;
            runLatch := FALSE;
            step := 90;

        ELSIF NOT vfdReady THEN
            deviceState := 'Stopping: drive not ready';
            vfdStartCmdOut := FALSE;
            runLatch := FALSE;
            step := 90;

        ELSIF NOT vfdRunFeedback THEN
            deviceState := 'Stopping: RUN feedback lost';
            vfdStartCmdOut := FALSE;
            runLatch := FALSE;
            step := 90;

        // Interlocks → normal stop
        ELSIF anyInterlockOpen THEN
            deviceState := 'Stopping: interlock open';
            vfdStartCmdOut := FALSE;
            runLatch := FALSE;
            step := 90;

        // Start toggled OFF while running => stop
        ELSIF NOT runLatch THEN
            deviceState := 'Stopping (Start toggled off)';
            vfdStartCmdOut := FALSE;
            step := 90;

        ELSE
            // ---- Input filtering (PT1) ----
            IF enableInputFilter THEN
                instPT1(in := whiteWaterSiloLevel, T := inputFilterTime, K := inputFilterGainK, out => pvEngFiltered);
            ELSE
                pvEngFiltered := whiteWaterSiloLevel;
            END_IF

